// unit & equipment number ---------------------------------------------------
      L     DB1400.DBW    0;
      T     #UnitNo;

      L     DB1405.DBW   14;
      L     1000;
      *I    ;
      L     #UnitNo;
      +I    ;
      T     #EquipmentID;

// CIP ----------------------------------------------------------------------
      L     DB1405.DBW   18;
      L     0;
      <I    ;
      =     #CIP;

// Communicating Units-------------------------------------------------------
      L     DB1405.DBD   10;
      L     DB1405.DBD  106;
      ==D   ;
      =     #ComCIP;

// emergency OK -------------------------------------------------------------
      A     DB1405.DBX   75.0; //General Emergency Stop OK
      =     #EStopOK;

NETWORK
TITLE =read other unit's data

      SET   ;

// ... General Unit ----------/

      CALL FC   563 (
           ActReq                   := M    101.0,
           PLCNo                    := DB1405.DBW   14,
           SourceUnitNo             := 99,
           IsTUnit                  := FALSE,
           DstComDRec               := DB1405.GEN,

           RET_VAL                  := #wRetVal);

// ... CIP Unit ------------- /

      CALL FC   563 (
           ActReq                   := M    101.0,
           PLCNo                    := 1,
           SourceUnitNo             := 71,
           IsTUnit                  := FALSE,
           DstComDRec               := DB1405.CIP,

           RET_VAL                  := #wRetVal);


NETWORK
TITLE =remote start

      SET   ;
// !!! insert correct condition of unit start !!!
      A     DB1401.DBX   15.0;
      A     DB1401.DBX   17.4;
      CLR   ;
      JCN   Strt;
      L     DB1405.DBD   10;
//L        L#-1;                            // Prid negative to start on its own
      T     #Prid;

      CALL FC    48 (
           UnitNo                   := #UnitNo,
           PrId                     := #Prid,
           Run                      := DB1401.DBX   17.4,
           PrIdTransfer             := TRUE,
           Start                    := TRUE,
           RetVal                   := #wRetVal);
Strt: NOP   0;
NETWORK
TITLE =external releases

      SET   ;
NETWORK
TITLE =write own unit data

      SET   ;

//-- CIP Communication ---------------------------------------
      AN    DB1401.DBX   15.0;
//      AN "U040SeqD".Seq.PO.B30 // CIP Active (Slave)
      A     #ComCIP;
      JCN   NCIP;
//Conductivity CIP Return
      L     DB1405.DBD  150;
      T     DB1401.DBD  626;

//Temperature CIP Return
      L     DB1405.DBD  146;
      T     DB1401.DBD  594;

//CIP Prerun Pump SP

      CALL FC    45 (
           SFM                      := DB1401.DBD  686,

           Indexes                  := #SFM36);

      L     0.000000e+000;
      A     #SFM36.I01;
      =     DB1405.DBX  171.7;
      JCN   pfc;
      L     DB1401.DBD  654;
pfc:  NOP   0;
      A     #SFM36.I02;
      =     DB1405.DBX  172.0;
      JCN   ppc;
      L     DB1401.DBD  670;
ppc:  NOP   0;
      A     #SFM36.I03;
      =     DB1405.DBX  171.6;
      JCN   pxc;
      L     DB1401.DBD  574;
pxc:  NOP   0;
      T     DB1405.DBD  182;

//CIP Return
      L     DB1401.DBD  558;
      T     DB1405.DBD  186;
      L     DB1405.DBD  138;
      T     DB1401.DBD  562;

//CIP Prerun
      L     DB1401.DBD  542;
      T     DB1405.DBD  190;
      L     DB1405.DBD  142;
      T     DB1401.DBD  546;

// Write Own Data to CIP
      L     DB1405.DBD   10;
      T     DB1405.DBD  154;

      L     DB1405.DBW   14;
      T     DB1405.DBW  158;

      L     DB1405.DBW   16;
      T     DB1405.DBW  160;

      L     DB1405.DBW   18;
      T     DB1405.DBW  162;

      L     DB1405.DBW   20;
      T     DB1405.DBW  164;

      L     DB1405.DBW   22;
      T     DB1405.DBW  166;

      A     DB1405.DBX   24.0;
      =     DB1405.DBX  168.0;

      A     DB1405.DBX   24.1;
      =     DB1405.DBX  168.1;

      A     DB1405.DBX   24.2;
      =     DB1405.DBX  168.2;

      A     DB1405.DBX   24.3;
      =     DB1405.DBX  168.3;

      A     DB1405.DBX   24.4;
      =     DB1405.DBX  168.4;

      A     DB1405.DBX   24.5;
      =     DB1405.DBX  168.5;

      A     DB1405.DBX   24.6;
      =     DB1405.DBX  168.6;

      A     DB1405.DBX   24.7;
      =     DB1405.DBX  168.7;

// Copy Data to CIP
      CALL SFC   20 (
           SRCBLK                   := DB1405.ToCIP,
           RET_VAL                  := #iRetVal,
           DSTBLK                   := DB1405.ToCIP);

NCIP: NOP   0;

//Empty Signal
//A     "U040SpID".SpI.Sig //!!!! Insert correct Empty Signal !!!
      CLR   ;
      =     DB1405.DBX   26.5;

//Full Signal
//A     "U040SpID".SpI.Sig //!!!! Insert correct Full Signal !!!
      CLR   ;
      =     DB1405.DBX   26.2;

//CIP Program Selected
      A     #CIP;
      =     DB1405.DBX   27.1;

// Emergency Stop
      A     #EStopOK; //If needed add or replace with own SpI
      =     DB1405.DBX   27.0; //Emergency Stop OK


NETWORK
TITLE = read from other unit data

END_FUNCTION_BLOCK

FUNCTION_BLOCK FB 1409
TITLE =U040: Water Treatment General
AUTHOR : Woermann
FAMILY : BOTEC_F1
NAME : Sim
VERSION : 0.1


VAR_TEMP
  CIP : BOOL ;	//CIP active
  xTmp : BOOL ;	//Temporary BOOL (free for general use)
  iTmp : INT ;	//Temporary INT (free for general use)
  rTmp : REAL ;	//Temporary REAL (free for general use)
  UnitNo : INT ;	//Unit Number
END_VAR
BEGIN
NETWORK
TITLE =General

      SET   ;
// get unit number ----------------------------------------------------------
      L     DB1400.DBW    0;
      T     #UnitNo;

// CIP ----------------------------------------------------------------------
      L     DB1401.DBD   54;
      L     0;
      <D    ;
      =     #CIP;

NETWORK
TITLE =Actuator

      A     DB1401.DBX   17.3;

NETWORK
TITLE =Special Input

      A     DB1401.DBX   17.3;
      =     DB2401.DBX   81.3;
      =     DB2401.DBX  141.3;
      =     DB2401.DBX  201.3;
      =     DB2401.DBX  261.3;
      =     DB2401.DBX  321.3;
      =     DB2401.DBX  381.3;

NETWORK
TITLE =Counter

      A     DB1401.DBX   17.3;
      A     M    101.0;


      CLR   ;
NETWORK
TITLE =Analog Input

      A     DB1401.DBX   17.3;

NETWORK
TITLE =Universal Value

      A     DB1401.DBX   17.3;
//      =     "U040UnVD".unv001.Sim;
//      =     "U040UnVD".unv002.Sim;

NETWORK
TITLE =PID

      A     DB1401.DBX   17.3;

NETWORK
TITLE =Message

      A     DB1401.DBX   17.3;
//      =     "U040MsgD".msg001.Sim;
//      =     "U040MsgD".msg002.Sim;

NETWORK
TITLE =VLT

      A     DB1401.DBX   17.3;

END_FUNCTION_BLOCK

FUNCTION_BLOCK FB 1435
TITLE =U043: Water Transfer Plant 3
FAMILY : BOTEC_F1
NAME : Comm
VERSION : 0.1


VAR_TEMP
  iRetVal : INT ;	//return value as integer
  wRetVal : WORD ;	//return value as word
  Run : BOOL ;	//Unit in "RUN" mode
  EStopOK : BOOL ;	//Emergency Stop OK
  CIP : BOOL ;	//CIP Program Selected
  ComCIP : BOOL ;	//Communication with CIP Active
  xTmp : BOOL ;	//Temporary BOOL (free for general use)
  iTmp : INT ;	//Temporary INT (free for general use)
  rTmp : REAL ;	//Temporary REAL (free for general use)
  dTmp : DINT ;	//Temporary DINT (free for general use)
  UnitNo : INT ;	//Unit Number
  EquipmentID : INT ;	//Equipment ID
  Prid : DINT ;	//Process ID
  SFM36 : STRUCT 	// CIP Pump Mode
   I00 : BOOL ;	// Off
   I01 : BOOL ;	// Flow
   I02 : BOOL ;	// Pressure
   I03 : BOOL ;	// Fix Speed
   I04 : BOOL ;
   I05 : BOOL ;
   I06 : BOOL ;
   I07 : BOOL ;
   I08 : BOOL ;
   I09 : BOOL ;
   I10 : BOOL ;
   I11 : BOOL ;
   I12 : BOOL ;
   I13 : BOOL ;
   I14 : BOOL ;
   I15 : BOOL ;
   I16 : BOOL ;
   I17 : BOOL ;
   I18 : BOOL ;
   I19 : BOOL ;
   I20 : BOOL ;
   I21 : BOOL ;
   I22 : BOOL ;
   I23 : BOOL ;
   I24 : BOOL ;
   I25 : BOOL ;
   I26 : BOOL ;
   I27 : BOOL ;
   I28 : BOOL ;
   I29 : BOOL ;
   I30 : BOOL ;
   I31 : BOOL ;
  END_STRUCT ;
END_VAR
BEGIN
NETWORK
TITLE =general

      SET   ;

// unit & equipment number ---------------------------------------------------
      L     DB1430.DBW    0;
      T     #UnitNo;

      L     DB1435.DBW   14;
      L     1000;
      *I    ;
      L     #UnitNo;
      +I    ;
      T     #EquipmentID;

// CIP ----------------------------------------------------------------------
      L     DB1435.DBW   18;
      L     0;
      <I    ;
      =     #CIP;

// Communicating Units-------------------------------------------------------
      L     DB1435.DBD   10;
      L     DB1435.DBD  106;
      ==D   ;
      =     #ComCIP;

// emergency OK -------------------------------------------------------------
      A     DB1435.DBX   75.0; //General Emergency Stop OK
      =     #EStopOK;

NETWORK
TITLE =read other unit's data

      SET   ;

// ... General Unit ----------/

      CALL FC   563 (
           ActReq                   := M    101.0,
           PLCNo                    := DB1435.DBW   14,
           SourceUnitNo             := 99,
           IsTUnit                  := FALSE,
           DstComDRec               := DB1435.GEN,
           RET_VAL                  := #wRetVal);


// ... CIP Unit ------------- /

      CALL FC   563 (
           ActReq                   := M    101.0,
           PLCNo                    := 1,
           SourceUnitNo             := 71,
           IsTUnit                  := FALSE,
           DstComDRec               := DB1435.CIP,
           RET_VAL                  := #wRetVal);



NETWORK
TITLE =remote start

      SET   ;
// !!! insert correct condition of unit start !!!
      A     DB1431.DBX   15.0;
      A     DB1431.DBX   17.4;
      CLR   ;
      JCN   Strt;
      L     L#-1; // Prid negative to start on its own
      T     #Prid;

      CALL FC    48 (
           UnitNo                   := #UnitNo,
           PrId                     := #Prid,
           Run                      := DB1431.DBX   17.4,
           PrIdTransfer             := TRUE,
           Start                    := TRUE,
           RetVal                   := #wRetVal);
Strt: NOP   0;
NETWORK
TITLE =external releases

      SET   ;
      =     DB2430.DBX  186.7;
      =     DB2430.DBX  266.7;
      =     DB2430.DBX  346.7;
NETWORK
TITLE =write own unit data

      SET   ;

//-- CIP Communication ---------------------------------------
      AN    DB1431.DBX   15.0;
//      AN "U043SeqD".Seq.PO.B30 // CIP Active (Slave)
      A     #ComCIP;
      JCN   NCIP;
//Conductivity CIP Return
      L     DB1435.DBD  150;
      T     DB1431.DBD  626;

//Temperature CIP Return
      L     DB1435.DBD  146;
      T     DB1431.DBD  594;

//CIP Prerun Pump SP

      CALL FC    45 (
           SFM                      := DB1431.DBD  686,
           Indexes                  := #SFM36);


      L     0.000000e+000;
      A     #SFM36.I01;
      =     DB1435.DBX  171.7;
      JCN   pfc;
      L     DB1431.DBD  654;
pfc:  NOP   0;
      A     #SFM36.I02;
      =     DB1435.DBX  172.0;
      JCN   ppc;
      L     DB1431.DBD  670;
ppc:  NOP   0;
      A     #SFM36.I03;
      =     DB1435.DBX  171.6;
      JCN   pxc;
      L     DB1431.DBD  574;
pxc:  NOP   0;
      T     DB1435.DBD  182;

//CIP Return
      L     DB1431.DBD  558;
      T     DB1435.DBD  186;
      L     DB1435.DBD  138;
      T     DB1431.DBD  562;

//CIP Prerun
      L     DB1431.DBD  542;
      T     DB1435.DBD  190;
      L     DB1435.DBD  142;
      T     DB1431.DBD  546;

// Write Own Data to CIP
      L     DB1435.DBD   10;
      T     DB1435.DBD  154;

      L     DB1435.DBW   14;
      T     DB1435.DBW  158;

      L     DB1435.DBW   16;
      T     DB1435.DBW  160;

      L     DB1435.DBW   18;
      T     DB1435.DBW  162;

      L     DB1435.DBW   20;
      T     DB1435.DBW  164;

      L     DB1435.DBW   22;
      T     DB1435.DBW  166;

      A     DB1435.DBX   24.0;
      =     DB1435.DBX  168.0;

      A     DB1435.DBX   24.1;
      =     DB1435.DBX  168.1;

      A     DB1435.DBX   24.2;
      =     DB1435.DBX  168.2;

      A     DB1435.DBX   24.3;
      =     DB1435.DBX  168.3;

      A     DB1435.DBX   24.4;
      =     DB1435.DBX  168.4;

      A     DB1435.DBX   24.5;
      =     DB1435.DBX  168.5;

      A     DB1435.DBX   24.6;
      =     DB1435.DBX  168.6;

      A     DB1435.DBX   24.7;
      =     DB1435.DBX  168.7;

// Copy Data to CIP
      CALL SFC   20 (
           SRCBLK                   := DB1435.ToCIP,
           RET_VAL                  := #iRetVal,
           DSTBLK                   := DB1435.ToCIP);

NCIP: NOP   0;

//Empty Signal
//A     "U043SpID".SpI.Sig //!!!! Insert correct Empty Signal !!!
      CLR   ;
      =     DB1435.DBX   26.5;

//Full Signal
//A     "U043SpID".SpI.Sig //!!!! Insert correct Full Signal !!!
      CLR   ;
      =     DB1435.DBX   26.2;

//CIP Program Selected
      A     #CIP;
      =     DB1435.DBX   27.1;

// Emergency Stop
      A     #EStopOK; //If needed add or replace with own SpI
      =     DB1435.DBX   27.0; //Emergency Stop OK



NETWORK
TITLE = read from other unit data



END_FUNCTION_BLOCK

FUNCTION_BLOCK FB 1439
TITLE =U043: Water Transfer Plant 3
AUTHOR : Woermann
FAMILY : BOTEC_F1
NAME : Sim
VERSION : 0.1


VAR_TEMP
  CIP : BOOL ;	//CIP active
  xTmp : BOOL ;	//Temporary BOOL (free for general use)
  iTmp : INT ;	//Temporary INT (free for general use)
  rTmp : REAL ;	//Temporary REAL (free for general use)
  UnitNo : INT ;	//Unit Number
END_VAR
BEGIN
NETWORK
TITLE =General

      SET   ;
// get unit number ----------------------------------------------------------
      L     DB1430.DBW    0;
      T     #UnitNo;

// CIP ----------------------------------------------------------------------
      L     DB1431.DBD   54;
      L     0;
      <D    ;
      =     #CIP;

NETWORK
TITLE =Actuator

      A     DB1431.DBX   17.3;
      =     DB2430.DBX  185.3;
      =     DB2430.DBX  265.3;
      =     DB2430.DBX  345.3;

NETWORK
TITLE =Special Input

      A     DB1431.DBX   17.3;
      =     DB2431.DBX   81.3;

NETWORK
TITLE =Counter

      A     DB1431.DBX   17.3;
      A     M    101.0;


      CLR   ;
NETWORK
TITLE =Analog Input

      A     DB1431.DBX   17.3;

NETWORK
TITLE =Universal Value

      A     DB1431.DBX   17.3;
//      =     "U043UnVD".unv001.Sim;
//      =     "U043UnVD".unv002.Sim;
//      =     "U043UnVD".unv003.Sim;
//      =     "U043UnVD".unv004.Sim;

NETWORK
TITLE =PID

      A     DB1431.DBX   17.3;

NETWORK
TITLE =Message

      A     DB1431.DBX   17.3;
//      =     "U043MsgD".msg001.Sim;
//      =     "U043MsgD".msg002.Sim;
//      =     "U043MsgD".msg003.Sim;

NETWORK
TITLE =VLT

      A     DB1431.DBX   17.3;

END_FUNCTION_BLOCK

FUNCTION_BLOCK FB 1455
TITLE =U045: Water Transfer Plant 5
FAMILY : BOTEC_F1
NAME : Comm
VERSION : 0.1


VAR_TEMP
  iRetVal : INT ;	//return value as integer
  wRetVal : WORD ;	//return value as word
  Run : BOOL ;	//Unit in "RUN" mode
  EStopOK : BOOL ;	//Emergency Stop OK
  CIP : BOOL ;	//CIP Program Selected
  ComCIP : BOOL ;	//Communication with CIP Active
  xTmp : BOOL ;	//Temporary BOOL (free for general use)
  iTmp : INT ;	//Temporary INT (free for general use)
  rTmp : REAL ;	//Temporary REAL (free for general use)
  dTmp : DINT ;	//Temporary DINT (free for general use)
  UnitNo : INT ;	//Unit Number
  EquipmentID : INT ;	//Equipment ID
  Prid : DINT ;	//Process ID
  SFM36 : STRUCT 	// CIP Pump Mode
   I00 : BOOL ;	// Off
   I01 : BOOL ;	// Flow
   I02 : BOOL ;	// Pressure
   I03 : BOOL ;	// Fix Speed
   I04 : BOOL ;
   I05 : BOOL ;
   I06 : BOOL ;
   I07 : BOOL ;
   I08 : BOOL ;
   I09 : BOOL ;
   I10 : BOOL ;
   I11 : BOOL ;
   I12 : BOOL ;
   I13 : BOOL ;
   I14 : BOOL ;
   I15 : BOOL ;
   I16 : BOOL ;
   I17 : BOOL ;
   I18 : BOOL ;
   I19 : BOOL ;
   I20 : BOOL ;
   I21 : BOOL ;
   I22 : BOOL ;
   I23 : BOOL ;
   I24 : BOOL ;
   I25 : BOOL ;
   I26 : BOOL ;
   I27 : BOOL ;
   I28 : BOOL ;
   I29 : BOOL ;
   I30 : BOOL ;
   I31 : BOOL ;
  END_STRUCT ;
  SRCUnit : INT ;	//Source Water Tank
  DummyBool : BOOL ;
END_VAR
BEGIN
NETWORK
TITLE =general

      SET   ;

// unit & equipment number ---------------------------------------------------
      L     DB1450.DBW    0;
      T     #UnitNo;

      L     DB1455.DBW   14;
      L     1000;
      *I    ;
      L     #UnitNo;
      +I    ;
      T     #EquipmentID;

// CIP ----------------------------------------------------------------------
      L     DB1455.DBW   18;
      L     0;
      <I    ;
      =     #CIP;

// Communicating Units-------------------------------------------------------
      L     DB1455.DBD   10;
      L     DB1455.DBD  106;
      ==D   ;
      =     #ComCIP;

// emergency OK -------------------------------------------------------------
      A     DB1455.DBX   75.0; //General Emergency Stop OK
      =     #EStopOK;

NETWORK
TITLE =remote start

      SET   ;
      L     DB1455.DBD   10;

// !!! insert correct condition of unit start !!!
      A     DB1451.DBX   15.0;
      A     DB1451.DBX   17.4;
      CLR   ;
      JCN   Strt;
      L     DB1455.DBD   10;
//L        L#-1;                            // Prid negative to start on its own
      T     #Prid;

      CALL FC    48 (
           UnitNo                   := #UnitNo,
           PrId                     := #Prid,
           Run                      := DB1451.DBX   17.4,
           PrIdTransfer             := TRUE,
           Start                    := TRUE,
           RetVal                   := #wRetVal);
Strt: NOP   0;
END_FUNCTION_BLOCK

FUNCTION_BLOCK FB 1459
TITLE =U045: Water Transfer Plant 5
AUTHOR : Woermann
FAMILY : BOTEC_F1
NAME : Sim
VERSION : 0.1


VAR_TEMP
  CIP : BOOL ;	//CIP active
  xTmp : BOOL ;	//Temporary BOOL (free for general use)
  iTmp : INT ;	//Temporary INT (free for general use)
  rTmp : REAL ;	//Temporary REAL (free for general use)
  UnitNo : INT ;	//Unit Number
END_VAR
BEGIN
NETWORK
TITLE =General

      SET   ;
// get unit number ----------------------------------------------------------
      L     DB1450.DBW    0;
      T     #UnitNo;

// CIP ----------------------------------------------------------------------
      L     DB1451.DBD   54;
      L     0;
      <D    ;
      =     #CIP;

NETWORK
TITLE =Actuator

      A     DB1451.DBX   17.3;
      =     DB2450.DBX  425.3;
      =     DB2450.DBX  505.3;
      =     DB2450.DBX  585.3;
      =     DB2450.DBX  665.3;

NETWORK
TITLE =Special Input

      A     DB1451.DBX   17.3;

NETWORK
TITLE =Counter

      A     DB1451.DBX   17.3;
      A     M    101.0;


      CLR   ;
NETWORK
TITLE =Analog Input

      A     DB1451.DBX   17.3;

NETWORK
TITLE =Universal Value

      A     DB1451.DBX   17.3;
//      =     "U045UnVD".unv001.Sim;
//      =     "U045UnVD".unv002.Sim;
//      =     "U045UnVD".unv003.Sim;
//      =     "U045UnVD".unv004.Sim;

NETWORK
TITLE =PID

      A     DB1451.DBX   17.3;

NETWORK
TITLE =Message

      A     DB1451.DBX   17.3;
//      =     "U045MsgD".msg001.Sim;
//      =     "U045MsgD".msg002.Sim;
//      =     "U045MsgD".msg003.Sim;

NETWORK
TITLE =VLT

      A     DB1451.DBX   17.3;

END_FUNCTION_BLOCK

FUNCTION_BLOCK FB 1475
TITLE =U047: Water Transfer Plant 7
FAMILY : BOTEC_F1
NAME : Comm
VERSION : 0.1


VAR_TEMP
  iRetVal : INT ;	//return value as integer
  wRetVal : WORD ;	//return value as word
  Run : BOOL ;	//Unit in "RUN" mode
  EStopOK : BOOL ;	//Emergency Stop OK
  CIP : BOOL ;	//CIP Program Selected
  ComCIP : BOOL ;	//Communication with CIP Active
  xTmp : BOOL ;	//Temporary BOOL (free for general use)
  iTmp : INT ;	//Temporary INT (free for general use)
  rTmp : REAL ;	//Temporary REAL (free for general use)
  dTmp : DINT ;	//Temporary DINT (free for general use)
  UnitNo : INT ;	//Unit Number
  EquipmentID : INT ;	//Equipment ID
  Prid : DINT ;	//Process ID
  SFM36 : STRUCT 	// CIP Pump Mode
   I00 : BOOL ;	// Off
   I01 : BOOL ;	// Flow
   I02 : BOOL ;	// Pressure
   I03 : BOOL ;	// Fix Speed
   I04 : BOOL ;
   I05 : BOOL ;
   I06 : BOOL ;
   I07 : BOOL ;
   I08 : BOOL ;
   I09 : BOOL ;
   I10 : BOOL ;
   I11 : BOOL ;
   I12 : BOOL ;
   I13 : BOOL ;
   I14 : BOOL ;
   I15 : BOOL ;
   I16 : BOOL ;
   I17 : BOOL ;
   I18 : BOOL ;
   I19 : BOOL ;
   I20 : BOOL ;
   I21 : BOOL ;
   I22 : BOOL ;
   I23 : BOOL ;
   I24 : BOOL ;
   I25 : BOOL ;
   I26 : BOOL ;
   I27 : BOOL ;
   I28 : BOOL ;
   I29 : BOOL ;
   I30 : BOOL ;
   I31 : BOOL ;
  END_STRUCT ;
END_VAR
BEGIN
NETWORK
TITLE =general

      SET   ;

// unit & equipment number ---------------------------------------------------
      L     DB1470.DBW    0;
      T     #UnitNo;

      L     DB1475.DBW   14;
      L     1000;
      *I    ;
      L     #UnitNo;
      +I    ;
      T     #EquipmentID;

// CIP ----------------------------------------------------------------------
      L     DB1475.DBW   18;
      L     0;
      <I    ;
      =     #CIP;

// Communicating Units-------------------------------------------------------
      L     DB1475.DBD   10;
      L     DB1475.DBD  106;
      ==D   ;
      =     #ComCIP;

// emergency OK -------------------------------------------------------------
      A     DB1475.DBX   75.0; //General Emergency Stop OK
      =     #EStopOK;

NETWORK
TITLE =read other unit's data

      SET   ;

// ... General Unit ----------/

      CALL FC   563 (
           ActReq                   := M    101.0,
           PLCNo                    := DB1475.DBW   14,
           SourceUnitNo             := 99,
           IsTUnit                  := FALSE,
           DstComDRec               := DB1475.GEN,
           RET_VAL                  := #wRetVal);


NETWORK
TITLE =remote start

      SET   ;
// !!! insert correct condition of unit start !!!
      A     DB1471.DBX   15.0;
      A     DB1471.DBX   17.4;
      CLR   ;
      JCN   Strt;
      L     DB1475.DBD   10;
//L        L#-1;                            // Prid negative to start on its own
      T     #Prid;

      CALL FC    48 (
           UnitNo                   := #UnitNo,
           PrId                     := #Prid,
           Run                      := DB1471.DBX   17.4,
           PrIdTransfer             := TRUE,
           Start                    := TRUE,
           RetVal                   := #wRetVal);
Strt: NOP   0;
NETWORK
TITLE =external releases

      SET   ;
      =     DB2470.DBX  186.7;
      =     DB2470.DBX  266.7;
      =     DB2470.DBX  346.7;
      =     DB2470.DBX  426.7;
      =     DB2470.DBX  506.7;
      =     DB2470.DBX  586.7;
      =     DB2470.DBX  666.7;
NETWORK
TITLE =write own unit data

      SET   ;

//-- CIP Communication ---------------------------------------
      AN    DB1471.DBX   15.0;
//      AN "U047SeqD".Seq.PO.B30 // CIP Active (Slave)
      A     #ComCIP;
      JCN   NCIP;
//Conductivity CIP Return
      L     DB1475.DBD  150;
      T     DB1471.DBD  626;

//Temperature CIP Return
      L     DB1475.DBD  146;
      T     DB1471.DBD  594;

//CIP Prerun Pump SP

      CALL FC    45 (
           SFM                      := DB1471.DBD  686,
           Indexes                  := #SFM36);


      L     0.000000e+000;
      A     #SFM36.I01;
      =     DB1475.DBX  171.7;
      JCN   pfc;
      L     DB1471.DBD  654;
pfc:  NOP   0;
      A     #SFM36.I02;
      =     DB1475.DBX  172.0;
      JCN   ppc;
      L     DB1471.DBD  670;
ppc:  NOP   0;
      A     #SFM36.I03;
      =     DB1475.DBX  171.6;
      JCN   pxc;
      L     DB1471.DBD  574;
pxc:  NOP   0;
      T     DB1475.DBD  182;

//CIP Return
      L     DB1471.DBD  558;
      T     DB1475.DBD  186;
      L     DB1475.DBD  138;
      T     DB1471.DBD  562;

//CIP Prerun
      L     DB1471.DBD  542;
      T     DB1475.DBD  190;
      L     DB1475.DBD  142;
      T     DB1471.DBD  546;

// Write Own Data to CIP
      L     DB1475.DBD   10;
      T     DB1475.DBD  154;

      L     DB1475.DBW   14;
      T     DB1475.DBW  158;

      L     DB1475.DBW   16;
      T     DB1475.DBW  160;

      L     DB1475.DBW   18;
      T     DB1475.DBW  162;

      L     DB1475.DBW   20;
      T     DB1475.DBW  164;

      L     DB1475.DBW   22;
      T     DB1475.DBW  166;

      A     DB1475.DBX   24.0;
      =     DB1475.DBX  168.0;

      A     DB1475.DBX   24.1;
      =     DB1475.DBX  168.1;

      A     DB1475.DBX   24.2;
      =     DB1475.DBX  168.2;

      A     DB1475.DBX   24.3;
      =     DB1475.DBX  168.3;

      A     DB1475.DBX   24.4;
      =     DB1475.DBX  168.4;

      A     DB1475.DBX   24.5;
      =     DB1475.DBX  168.5;

      A     DB1475.DBX   24.6;
      =     DB1475.DBX  168.6;

      A     DB1475.DBX   24.7;
      =     DB1475.DBX  168.7;

// Copy Data to CIP
      CALL SFC   20 (
           SRCBLK                   := DB1475.ToCIP,
           RET_VAL                  := #iRetVal,
           DSTBLK                   := DB1475.ToCIP);

NCIP: NOP   0;

//Empty Signal
//A     "U047SpID".SpI.Sig //!!!! Insert correct Empty Signal !!!
      CLR   ;
      =     DB1475.DBX   26.5;

//Full Signal
//A     "U047SpID".SpI.Sig //!!!! Insert correct Full Signal !!!
      CLR   ;
      =     DB1475.DBX   26.2;

//CIP Program Selected
      A     #CIP;
      =     DB1475.DBX   27.1;

// Emergency Stop
      A     #EStopOK; //If needed add or replace with own SpI
      =     DB1475.DBX   27.0; //Emergency Stop OK


NETWORK
TITLE = read from other unit data



END_FUNCTION_BLOCK

FUNCTION_BLOCK FB 1479
TITLE =U047: Water Transfer Plant 7
AUTHOR : Woermann
FAMILY : BOTEC_F1
NAME : Sim
VERSION : 0.1


VAR_TEMP
  CIP : BOOL ;	//CIP active
  xTmp : BOOL ;	//Temporary BOOL (free for general use)
  iTmp : INT ;	//Temporary INT (free for general use)
  rTmp : REAL ;	//Temporary REAL (free for general use)
  UnitNo : INT ;	//Unit Number
END_VAR
BEGIN
NETWORK
TITLE =General

      SET   ;
// get unit number ----------------------------------------------------------
      L     DB1470.DBW    0;
      T     #UnitNo;

// CIP ----------------------------------------------------------------------
      L     DB1471.DBD   54;
      L     0;
      <D    ;
      =     #CIP;

NETWORK
TITLE =Actuator

      A     DB1471.DBX   17.3;
      =     DB2470.DBX  185.3;
      =     DB2470.DBX  265.3;
      =     DB2470.DBX  345.3;
      =     DB2470.DBX  425.3;
      =     DB2470.DBX  505.3;
      =     DB2470.DBX  585.3;
      =     DB2470.DBX  665.3;

NETWORK
TITLE =Special Input

      A     DB1471.DBX   17.3;

NETWORK
TITLE =Counter

      A     DB1471.DBX   17.3;
      A     M    101.0;


      CLR   ;
NETWORK
TITLE =Analog Input

      A     DB1471.DBX   17.3;

NETWORK
TITLE =Universal Value

      A     DB1471.DBX   17.3;
//      =     "U047UnVD".unv001.Sim;
//      =     "U047UnVD".unv002.Sim;
//      =     "U047UnVD".unv003.Sim;
//      =     "U047UnVD".unv004.Sim;

NETWORK
TITLE =PID

      A     DB1471.DBX   17.3;

NETWORK
TITLE =Message

      A     DB1471.DBX   17.3;
//      =     "U047MsgD".msg001.Sim;
//      =     "U047MsgD".msg002.Sim;
//      =     "U047MsgD".msg003.Sim;

NETWORK
TITLE =VLT

      A     DB1471.DBX   17.3;

END_FUNCTION_BLOCK

FUNCTION_BLOCK FB 1485
TITLE =U048: Water Transfer Plant 8
FAMILY : BOTEC_F1
NAME : Comm
VERSION : 0.1


VAR_TEMP
  iRetVal : INT ;	//return value as integer
  wRetVal : WORD ;	//return value as word
  Run : BOOL ;	//Unit in "RUN" mode
  EStopOK : BOOL ;	//Emergency Stop OK
  CIP : BOOL ;	//CIP Program Selected
  ComCIP : BOOL ;	//Communication with CIP Active
  xTmp : BOOL ;	//Temporary BOOL (free for general use)
  iTmp : INT ;	//Temporary INT (free for general use)
  rTmp : REAL ;	//Temporary REAL (free for general use)
  dTmp : DINT ;	//Temporary DINT (free for general use)
  UnitNo : INT ;	//Unit Number
  EquipmentID : INT ;	//Equipment ID
  Prid : DINT ;	//Process ID
  SFM36 : STRUCT 	// CIP Pump Mode
   I00 : BOOL ;	// Off
   I01 : BOOL ;	// Flow
   I02 : BOOL ;	// Pressure
   I03 : BOOL ;	// Fix Speed
   I04 : BOOL ;
   I05 : BOOL ;
   I06 : BOOL ;
   I07 : BOOL ;
   I08 : BOOL ;
   I09 : BOOL ;
   I10 : BOOL ;
   I11 : BOOL ;
   I12 : BOOL ;
   I13 : BOOL ;
   I14 : BOOL ;
   I15 : BOOL ;
   I16 : BOOL ;
   I17 : BOOL ;
   I18 : BOOL ;
   I19 : BOOL ;
   I20 : BOOL ;
   I21 : BOOL ;
   I22 : BOOL ;
   I23 : BOOL ;
   I24 : BOOL ;
   I25 : BOOL ;
   I26 : BOOL ;
   I27 : BOOL ;
   I28 : BOOL ;
   I29 : BOOL ;
   I30 : BOOL ;
   I31 : BOOL ;
  END_STRUCT ;
END_VAR
BEGIN
NETWORK
TITLE =general

      SET   ;

// unit & equipment number ---------------------------------------------------
      L     DB1480.DBW    0;
      T     #UnitNo;

      L     DB1485.DBW   14;
      L     1000;
      *I    ;
      L     #UnitNo;
      +I    ;
      T     #EquipmentID;

// CIP ----------------------------------------------------------------------
      L     DB1485.DBW   18;
      L     0;
      <I    ;
      =     #CIP;

// Communicating Units-------------------------------------------------------
      L     DB1485.DBD   10;
      L     DB1485.DBD  106;
      ==D   ;
      =     #ComCIP;

// emergency OK -------------------------------------------------------------
      A     DB1485.DBX   75.0; //General Emergency Stop OK
      =     #EStopOK;

NETWORK
TITLE =read other unit's data

      SET   ;

// ... General Unit ----------/

      CALL FC   563 (
           ActReq                   := M    101.0,
           PLCNo                    := DB1485.DBW   14,
           SourceUnitNo             := 99,
           IsTUnit                  := FALSE,
           DstComDRec               := DB1485.GEN,
           RET_VAL                  := #wRetVal);

NETWORK
TITLE =remote start

      SET   ;
// !!! insert correct condition of unit start !!!
      A     DB1481.DBX   15.0;
      A     DB1481.DBX   17.4;
      CLR   ;
      JCN   Strt;
      L     DB1485.DBD   10;
//L        L#-1;                            // Prid negative to start on its own
      T     #Prid;

      CALL FC    48 (
           UnitNo                   := #UnitNo,
           PrId                     := #Prid,
           Run                      := DB1481.DBX   17.4,
           PrIdTransfer             := TRUE,
           Start                    := TRUE,
           RetVal                   := #wRetVal);
Strt: NOP   0;
NETWORK
TITLE =external releases

      SET   ;
      =     DB2480.DBX  426.7;
      =     DB2480.DBX  506.7;
      =     DB2480.DBX  586.7;
      =     DB2480.DBX  666.7;
NETWORK
TITLE =write own unit data

      SET   ;

//-- CIP Communication ---------------------------------------
      AN    DB1481.DBX   15.0;
//      AN "U048SeqD".Seq.PO.B30 // CIP Active (Slave)
      A     #ComCIP;
      JCN   NCIP;
//Conductivity CIP Return
      L     DB1485.DBD  150;
      T     DB1481.DBD  626;

//Temperature CIP Return
      L     DB1485.DBD  146;
      T     DB1481.DBD  594;

//CIP Prerun Pump SP

      CALL FC    45 (
           SFM                      := DB1481.DBD  686,
           Indexes                  := #SFM36);


      L     0.000000e+000;
      A     #SFM36.I01;
      =     DB1485.DBX  171.7;
      JCN   pfc;
      L     DB1481.DBD  654;
pfc:  NOP   0;
      A     #SFM36.I02;
      =     DB1485.DBX  172.0;
      JCN   ppc;
      L     DB1481.DBD  670;
ppc:  NOP   0;
      A     #SFM36.I03;
      =     DB1485.DBX  171.6;
      JCN   pxc;
      L     DB1481.DBD  574;
pxc:  NOP   0;
      T     DB1485.DBD  182;

//CIP Return
      L     DB1481.DBD  558;
      T     DB1485.DBD  186;
      L     DB1485.DBD  138;
      T     DB1481.DBD  562;

//CIP Prerun
      L     DB1481.DBD  542;
      T     DB1485.DBD  190;
      L     DB1485.DBD  142;
      T     DB1481.DBD  546;

// Write Own Data to CIP
      L     DB1485.DBD   10;
      T     DB1485.DBD  154;

      L     DB1485.DBW   14;
      T     DB1485.DBW  158;

      L     DB1485.DBW   16;
      T     DB1485.DBW  160;

      L     DB1485.DBW   18;
      T     DB1485.DBW  162;

      L     DB1485.DBW   20;
      T     DB1485.DBW  164;

      L     DB1485.DBW   22;
      T     DB1485.DBW  166;

      A     DB1485.DBX   24.0;
      =     DB1485.DBX  168.0;

      A     DB1485.DBX   24.1;
      =     DB1485.DBX  168.1;

      A     DB1485.DBX   24.2;
      =     DB1485.DBX  168.2;

      A     DB1485.DBX   24.3;
      =     DB1485.DBX  168.3;

      A     DB1485.DBX   24.4;
      =     DB1485.DBX  168.4;

      A     DB1485.DBX   24.5;
      =     DB1485.DBX  168.5;

      A     DB1485.DBX   24.6;
      =     DB1485.DBX  168.6;

      A     DB1485.DBX   24.7;
      =     DB1485.DBX  168.7;

// Copy Data to CIP
      CALL SFC   20 (
           SRCBLK                   := DB1485.ToCIP,
           RET_VAL                  := #iRetVal,
           DSTBLK                   := DB1485.ToCIP);

NCIP: NOP   0;

//Empty Signal
//A     "U048SpID".SpI.Sig //!!!! Insert correct Empty Signal !!!
      CLR   ;
      =     DB1485.DBX   26.5;

//Full Signal
//A     "U048SpID".SpI.Sig //!!!! Insert correct Full Signal !!!
      CLR   ;
      =     DB1485.DBX   26.2;

//CIP Program Selected
      A     #CIP;
      =     DB1485.DBX   27.1;

// Emergency Stop
      A     #EStopOK; //If needed add or replace with own SpI
      =     DB1485.DBX   27.0; //Emergency Stop OK


NETWORK
TITLE = read from other unit data



END_FUNCTION_BLOCK

FUNCTION_BLOCK FB 1489
TITLE =U048: Water Transfer Plant 8
AUTHOR : Woermann
FAMILY : BOTEC_F1
NAME : Sim
VERSION : 0.1


VAR_TEMP
  CIP : BOOL ;	//CIP active
  xTmp : BOOL ;	//Temporary BOOL (free for general use)
  iTmp : INT ;	//Temporary INT (free for general use)
  rTmp : REAL ;	//Temporary REAL (free for general use)
  UnitNo : INT ;	//Unit Number
END_VAR
BEGIN
NETWORK
TITLE =General

      SET   ;
// get unit number ----------------------------------------------------------
      L     DB1480.DBW    0;
      T     #UnitNo;

// CIP ----------------------------------------------------------------------
      L     DB1481.DBD   54;
      L     0;
      <D    ;
      =     #CIP;

NETWORK
TITLE =Actuator

      A     DB1481.DBX   17.3;
      =     DB2480.DBX  425.3;
      =     DB2480.DBX  505.3;
      =     DB2480.DBX  585.3;
      =     DB2480.DBX  665.3;

NETWORK
TITLE =Special Input

      A     DB1481.DBX   17.3;

NETWORK
TITLE =Counter

      A     DB1481.DBX   17.3;
      A     M    101.0;


      CLR   ;
NETWORK
TITLE =Analog Input

      A     DB1481.DBX   17.3;

NETWORK
TITLE =Universal Value

      A     DB1481.DBX   17.3;
//      =     "U048UnVD".unv001.Sim;
//      =     "U048UnVD".unv002.Sim;
//      =     "U048UnVD".unv003.Sim;
//      =     "U048UnVD".unv004.Sim;

NETWORK
TITLE =PID

      A     DB1481.DBX   17.3;

NETWORK
TITLE =Message

      A     DB1481.DBX   17.3;
//      =     "U048MsgD".msg001.Sim;
//      =     "U048MsgD".msg002.Sim;
//      =     "U048MsgD".msg003.Sim;

NETWORK
TITLE =VLT

      A     DB1481.DBX   17.3;

END_FUNCTION_BLOCK

FUNCTION_BLOCK FB 1495
TITLE =U049: Water Transfer Plant 9
FAMILY : BOTEC_F1
NAME : Comm
VERSION : 0.1


VAR_TEMP
  iRetVal : INT ;	//return value as integer
  wRetVal : WORD ;	//return value as word
  Run : BOOL ;	//Unit in "RUN" mode
  EStopOK : BOOL ;	//Emergency Stop OK
  CIP : BOOL ;	//CIP Program Selected
  ComCIP : BOOL ;	//Communication with CIP Active
  xTmp : BOOL ;	//Temporary BOOL (free for general use)
  iTmp : INT ;	//Temporary INT (free for general use)
  rTmp : REAL ;	//Temporary REAL (free for general use)
  dTmp : DINT ;	//Temporary DINT (free for general use)
  UnitNo : INT ;	//Unit Number
  EquipmentID : INT ;	//Equipment ID
  Prid : DINT ;	//Process ID
  SFM36 : STRUCT 	// CIP Pump Mode
   I00 : BOOL ;	// Off
   I01 : BOOL ;	// Flow
   I02 : BOOL ;	// Pressure
   I03 : BOOL ;	// Fix Speed
   I04 : BOOL ;
   I05 : BOOL ;
   I06 : BOOL ;
   I07 : BOOL ;
   I08 : BOOL ;
   I09 : BOOL ;
   I10 : BOOL ;
   I11 : BOOL ;
   I12 : BOOL ;
   I13 : BOOL ;
   I14 : BOOL ;
   I15 : BOOL ;
   I16 : BOOL ;
   I17 : BOOL ;
   I18 : BOOL ;
   I19 : BOOL ;
   I20 : BOOL ;
   I21 : BOOL ;
   I22 : BOOL ;
   I23 : BOOL ;
   I24 : BOOL ;
   I25 : BOOL ;
   I26 : BOOL ;
   I27 : BOOL ;
   I28 : BOOL ;
   I29 : BOOL ;
   I30 : BOOL ;
   I31 : BOOL ;
  END_STRUCT ;
END_VAR
BEGIN
NETWORK
TITLE =general

      SET   ;

// unit & equipment number ---------------------------------------------------
      L     DB1490.DBW    0;
      T     #UnitNo;

      L     DB1495.DBW   14;
      L     1000;
      *I    ;
      L     #UnitNo;
      +I    ;
      T     #EquipmentID;

// CIP ----------------------------------------------------------------------
      L     DB1495.DBW   18;
      L     0;
      <I    ;
      =     #CIP;

// Communicating Units-------------------------------------------------------
      L     DB1495.DBD   10;
      L     DB1495.DBD  106;
      ==D   ;
      =     #ComCIP;

// emergency OK -------------------------------------------------------------
      A     DB1495.DBX   75.0; //General Emergency Stop OK
      =     #EStopOK;

NETWORK
TITLE =read other unit's data

      SET   ;

// ... General Unit ----------/

      CALL FC   563 (
           ActReq                   := M    101.0,
           PLCNo                    := DB1495.DBW   14,
           SourceUnitNo             := 99,
           IsTUnit                  := FALSE,
           DstComDRec               := DB1495.GEN,
           RET_VAL                  := #wRetVal);

NETWORK
TITLE =remote start

      SET   ;
// !!! insert correct condition of unit start !!!
      A     DB1491.DBX   15.0;
      A     DB1491.DBX   17.4;
      CLR   ;
      JCN   Strt;
      L     DB1495.DBD   10;
//L        L#-1;                            // Prid negative to start on its own
      T     #Prid;

      CALL FC    48 (
           UnitNo                   := #UnitNo,
           PrId                     := #Prid,
           Run                      := DB1491.DBX   17.4,
           PrIdTransfer             := TRUE,
           Start                    := TRUE,
           RetVal                   := #wRetVal);
Strt: NOP   0;
NETWORK
TITLE =external releases

      SET   ;
      =     DB2490.DBX  186.7;
      =     DB2490.DBX  266.7;
      =     DB2490.DBX  346.7;
      =     DB2490.DBX  426.7;
      =     DB2490.DBX  506.7;
      =     DB2490.DBX  586.7;
      =     DB2490.DBX  666.7;
NETWORK
TITLE =write own unit data

      SET   ;

//-- CIP Communication ---------------------------------------
      AN    DB1491.DBX   15.0;
//      AN "U049SeqD".Seq.PO.B30 // CIP Active (Slave)
      A     #ComCIP;
      JCN   NCIP;
//Conductivity CIP Return
      L     DB1495.DBD  150;
      T     DB1491.DBD  626;

//Temperature CIP Return
      L     DB1495.DBD  146;
      T     DB1491.DBD  594;

//CIP Prerun Pump SP

      CALL FC    45 (
           SFM                      := DB1491.DBD  686,
           Indexes                  := #SFM36);


      L     0.000000e+000;
      A     #SFM36.I01;
      =     DB1495.DBX  171.7;
      JCN   pfc;
      L     DB1491.DBD  654;
pfc:  NOP   0;
      A     #SFM36.I02;
      =     DB1495.DBX  172.0;
      JCN   ppc;
      L     DB1491.DBD  670;
ppc:  NOP   0;
      A     #SFM36.I03;
      =     DB1495.DBX  171.6;
      JCN   pxc;
      L     DB1491.DBD  574;
pxc:  NOP   0;
      T     DB1495.DBD  182;

//CIP Return
      L     DB1491.DBD  558;
      T     DB1495.DBD  186;
      L     DB1495.DBD  138;
      T     DB1491.DBD  562;

//CIP Prerun
      L     DB1491.DBD  542;
      T     DB1495.DBD  190;
      L     DB1495.DBD  142;
      T     DB1491.DBD  546;

// Write Own Data to CIP
      L     DB1495.DBD   10;
      T     DB1495.DBD  154;

      L     DB1495.DBW   14;
      T     DB1495.DBW  158;

      L     DB1495.DBW   16;
      T     DB1495.DBW  160;

      L     DB1495.DBW   18;
      T     DB1495.DBW  162;

      L     DB1495.DBW   20;
      T     DB1495.DBW  164;

      L     DB1495.DBW   22;
      T     DB1495.DBW  166;

      A     DB1495.DBX   24.0;
      =     DB1495.DBX  168.0;

      A     DB1495.DBX   24.1;
      =     DB1495.DBX  168.1;

      A     DB1495.DBX   24.2;
      =     DB1495.DBX  168.2;

      A     DB1495.DBX   24.3;
      =     DB1495.DBX  168.3;

      A     DB1495.DBX   24.4;
      =     DB1495.DBX  168.4;

      A     DB1495.DBX   24.5;
      =     DB1495.DBX  168.5;

      A     DB1495.DBX   24.6;
      =     DB1495.DBX  168.6;

      A     DB1495.DBX   24.7;
      =     DB1495.DBX  168.7;

// Copy Data to CIP
      CALL SFC   20 (
           SRCBLK                   := DB1495.ToCIP,
           RET_VAL                  := #iRetVal,
           DSTBLK                   := DB1495.ToCIP);

NCIP: NOP   0;

//Empty Signal
//A     "U049SpID".SpI.Sig //!!!! Insert correct Empty Signal !!!
      CLR   ;
      =     DB1495.DBX   26.5;

//Full Signal
//A     "U049SpID".SpI.Sig //!!!! Insert correct Full Signal !!!
      CLR   ;
      =     DB1495.DBX   26.2;

//CIP Program Selected
      A     #CIP;
      =     DB1495.DBX   27.1;

// Emergency Stop
      A     #EStopOK; //If needed add or replace with own SpI
      =     DB1495.DBX   27.0; //Emergency Stop OK


NETWORK
TITLE = read from other unit data



END_FUNCTION_BLOCK

FUNCTION_BLOCK FB 1499
TITLE =U049: Water Transfer Plant 9
AUTHOR : Woermann
FAMILY : BOTEC_F1
NAME : Sim
VERSION : 0.1


VAR_TEMP
  CIP : BOOL ;	//CIP active
  xTmp : BOOL ;	//Temporary BOOL (free for general use)
  iTmp : INT ;	//Temporary INT (free for general use)
  rTmp : REAL ;	//Temporary REAL (free for general use)
  UnitNo : INT ;	//Unit Number
END_VAR
BEGIN
NETWORK
TITLE =General

      SET   ;
// get unit number ----------------------------------------------------------
      L     DB1490.DBW    0;
      T     #UnitNo;

// CIP ----------------------------------------------------------------------
      L     DB1491.DBD   54;
      L     0;
      <D    ;
      =     #CIP;

NETWORK
TITLE =Actuator

      A     DB1491.DBX   17.3;
      =     DB2490.DBX  185.3;
      =     DB2490.DBX  265.3;
      =     DB2490.DBX  345.3;
      =     DB2490.DBX  425.3;
      =     DB2490.DBX  505.3;
      =     DB2490.DBX  585.3;
      =     DB2490.DBX  665.3;

NETWORK
TITLE =Special Input

      A     DB1491.DBX   17.3;

NETWORK
TITLE =Counter

      A     DB1491.DBX   17.3;
      A     M    101.0;


      CLR   ;
NETWORK
TITLE =Analog Input

      A     DB1491.DBX   17.3;

NETWORK
TITLE =Universal Value

      A     DB1491.DBX   17.3;
//      =     "U049UnVD".unv001.Sim;
//      =     "U049UnVD".unv002.Sim;
//      =     "U049UnVD".unv003.Sim;
//      =     "U049UnVD".unv004.Sim;

NETWORK
TITLE =PID

      A     DB1491.DBX   17.3;

NETWORK
TITLE =Message

      A     DB1491.DBX   17.3;
//      =     "U049MsgD".msg001.Sim;
//      =     "U049MsgD".msg002.Sim;
//      =     "U049MsgD".msg003.Sim;

NETWORK
TITLE =VLT

      A     DB1491.DBX   17.3;

END_FUNCTION_BLOCK

FUNCTION_BLOCK FB 1505
TITLE =U050: Water Transfer Plant 10
FAMILY : BOTEC_F1
NAME : Comm
VERSION : 0.1


VAR_TEMP
  iRetVal : INT ;	//return value as integer
  wRetVal : WORD ;	//return value as word
  Run : BOOL ;	//Unit in "RUN" mode
  EStopOK : BOOL ;	//Emergency Stop OK
  CIP : BOOL ;	//CIP Program Selected
  ComCIP : BOOL ;	//Communication with CIP Active
  xTmp : BOOL ;	//Temporary BOOL (free for general use)
  iTmp : INT ;	//Temporary INT (free for general use)
  rTmp : REAL ;	//Temporary REAL (free for general use)
  dTmp : DINT ;	//Temporary DINT (free for general use)
  UnitNo : INT ;	//Unit Number
  EquipmentID : INT ;	//Equipment ID
  Prid : DINT ;	//Process ID
  SFM36 : STRUCT 	// CIP Pump Mode
   I00 : BOOL ;	// Off
   I01 : BOOL ;	// Flow
   I02 : BOOL ;	// Pressure
   I03 : BOOL ;	// Fix Speed
   I04 : BOOL ;
   I05 : BOOL ;
   I06 : BOOL ;
   I07 : BOOL ;
   I08 : BOOL ;
   I09 : BOOL ;
   I10 : BOOL ;
   I11 : BOOL ;
   I12 : BOOL ;
   I13 : BOOL ;
   I14 : BOOL ;
   I15 : BOOL ;
   I16 : BOOL ;
   I17 : BOOL ;
   I18 : BOOL ;
   I19 : BOOL ;
   I20 : BOOL ;
   I21 : BOOL ;
   I22 : BOOL ;
   I23 : BOOL ;
   I24 : BOOL ;
   I25 : BOOL ;
   I26 : BOOL ;
   I27 : BOOL ;
   I28 : BOOL ;
   I29 : BOOL ;
   I30 : BOOL ;
   I31 : BOOL ;
  END_STRUCT ;
END_VAR
BEGIN
NETWORK
TITLE =general

      SET   ;

// unit & equipment number ---------------------------------------------------
      L     DB1500.DBW    0;
      T     #UnitNo;

      L     DB1505.DBW   14;
      L     1000;
      *I    ;
      L     #UnitNo;
      +I    ;
      T     #EquipmentID;

// CIP ----------------------------------------------------------------------
      L     DB1505.DBW   18;
      L     0;
      <I    ;
      =     #CIP;

// Communicating Units-------------------------------------------------------
      L     DB1505.DBD   10;
      L     DB1505.DBD  106;
      ==D   ;
      =     #ComCIP;

// emergency OK -------------------------------------------------------------
      A     DB1505.DBX   75.0; //General Emergency Stop OK
      =     #EStopOK;

NETWORK
TITLE =read other unit's data

      SET   ;

// ... General Unit ----------/

      CALL FC   563 (
           ActReq                   := M    101.0,
           PLCNo                    := DB1505.DBW   14,
           SourceUnitNo             := 99,
           IsTUnit                  := FALSE,
           DstComDRec               := DB1505.GEN,
           RET_VAL                  := #wRetVal);

NETWORK
TITLE =remote start

      SET   ;
// !!! insert correct condition of unit start !!!
      A     DB1501.DBX   15.0;
      A     DB1501.DBX   17.4;
      CLR   ;
      JCN   Strt;
      L     DB1505.DBD   10;
//L        L#-1;                            // Prid negative to start on its own
      T     #Prid;

      CALL FC    48 (
           UnitNo                   := #UnitNo,
           PrId                     := #Prid,
           Run                      := DB1501.DBX   17.4,
           PrIdTransfer             := TRUE,
           Start                    := TRUE,
           RetVal                   := #wRetVal);
Strt: NOP   0;
NETWORK
TITLE =external releases

      SET   ;
      =     DB2500.DBX  186.7;
      =     DB2500.DBX  266.7;
      =     DB2500.DBX  346.7;
      =     DB2500.DBX  426.7;
      =     DB2500.DBX  506.7;
      =     DB2500.DBX  586.7;
      =     DB2500.DBX  666.7;
NETWORK
TITLE =write own unit data

      SET   ;

//-- CIP Communication ---------------------------------------
      AN    DB1501.DBX   15.0;
//      AN "U050SeqD".Seq.PO.B30 // CIP Active (Slave)
      A     #ComCIP;
      JCN   NCIP;
//Conductivity CIP Return
      L     DB1505.DBD  150;
      T     DB1501.DBD  626;

//Temperature CIP Return
      L     DB1505.DBD  146;
      T     DB1501.DBD  594;

//CIP Prerun Pump SP

      CALL FC    45 (
           SFM                      := DB1501.DBD  686,
           Indexes                  := #SFM36);


      L     0.000000e+000;
      A     #SFM36.I01;
      =     DB1505.DBX  171.7;
      JCN   pfc;
      L     DB1501.DBD  654;
pfc:  NOP   0;
      A     #SFM36.I02;
      =     DB1505.DBX  172.0;
      JCN   ppc;
      L     DB1501.DBD  670;
ppc:  NOP   0;
      A     #SFM36.I03;
      =     DB1505.DBX  171.6;
      JCN   pxc;
      L     DB1501.DBD  574;
pxc:  NOP   0;
      T     DB1505.DBD  182;

//CIP Return
      L     DB1501.DBD  558;
      T     DB1505.DBD  186;
      L     DB1505.DBD  138;
      T     DB1501.DBD  562;

//CIP Prerun
      L     DB1501.DBD  542;
      T     DB1505.DBD  190;
      L     DB1505.DBD  142;
      T     DB1501.DBD  546;

// Write Own Data to CIP
      L     DB1505.DBD   10;
      T     DB1505.DBD  154;

      L     DB1505.DBW   14;
      T     DB1505.DBW  158;

      L     DB1505.DBW   16;
      T     DB1505.DBW  160;

      L     DB1505.DBW   18;
      T     DB1505.DBW  162;

      L     DB1505.DBW   20;
      T     DB1505.DBW  164;

      L     DB1505.DBW   22;
      T     DB1505.DBW  166;

      A     DB1505.DBX   24.0;
      =     DB1505.DBX  168.0;

      A     DB1505.DBX   24.1;
      =     DB1505.DBX  168.1;

      A     DB1505.DBX   24.2;
      =     DB1505.DBX  168.2;

      A     DB1505.DBX   24.3;
      =     DB1505.DBX  168.3;

      A     DB1505.DBX   24.4;
      =     DB1505.DBX  168.4;

      A     DB1505.DBX   24.5;
      =     DB1505.DBX  168.5;

      A     DB1505.DBX   24.6;
      =     DB1505.DBX  168.6;

      A     DB1505.DBX   24.7;
      =     DB1505.DBX  168.7;

// Copy Data to CIP
      CALL SFC   20 (
           SRCBLK                   := DB1505.ToCIP,
           RET_VAL                  := #iRetVal,
           DSTBLK                   := DB1505.ToCIP);

NCIP: NOP   0;

//Empty Signal
//A     "U050SpID".SpI.Sig //!!!! Insert correct Empty Signal !!!
      CLR   ;
      =     DB1505.DBX   26.5;

//Full Signal
//A     "U050SpID".SpI.Sig //!!!! Insert correct Full Signal !!!
      CLR   ;
      =     DB1505.DBX   26.2;

//CIP Program Selected
      A     #CIP;
      =     DB1505.DBX   27.1;

// Emergency Stop
      A     #EStopOK; //If needed add or replace with own SpI
      =     DB1505.DBX   27.0; //Emergency Stop OK


NETWORK
TITLE = read from other unit data



END_FUNCTION_BLOCK

FUNCTION_BLOCK FB 1509
TITLE =U050: Water Transfer Plant 10
AUTHOR : Woermann
FAMILY : BOTEC_F1
NAME : Sim
VERSION : 0.1


VAR_TEMP
  CIP : BOOL ;	//CIP active
  xTmp : BOOL ;	//Temporary BOOL (free for general use)
  iTmp : INT ;	//Temporary INT (free for general use)
  rTmp : REAL ;	//Temporary REAL (free for general use)
  UnitNo : INT ;	//Unit Number
END_VAR
BEGIN
NETWORK
TITLE =General

      SET   ;
// get unit number ----------------------------------------------------------
      L     DB1500.DBW    0;
      T     #UnitNo;

// CIP ----------------------------------------------------------------------
      L     DB1501.DBD   54;
      L     0;
      <D    ;
      =     #CIP;

NETWORK
TITLE =Actuator

      A     DB1501.DBX   17.3;
      =     DB2500.DBX  185.3;
      =     DB2500.DBX  265.3;
      =     DB2500.DBX  345.3;
      =     DB2500.DBX  425.3;
      =     DB2500.DBX  505.3;
      =     DB2500.DBX  585.3;
      =     DB2500.DBX  665.3;

NETWORK
TITLE =Special Input

      A     DB1501.DBX   17.3;

NETWORK
TITLE =Counter

      A     DB1501.DBX   17.3;
      A     M    101.0;


      CLR   ;
NETWORK
TITLE =Analog Input

      A     DB1501.DBX   17.3;

NETWORK
TITLE =Universal Value

      A     DB1501.DBX   17.3;
//      =     "U050UnVD".unv001.Sim;
//      =     "U050UnVD".unv002.Sim;
//      =     "U050UnVD".unv003.Sim;
//      =     "U050UnVD".unv004.Sim;

NETWORK
TITLE =PID

      A     DB1501.DBX   17.3;

NETWORK
TITLE =Message

      A     DB1501.DBX   17.3;
//      =     "U050MsgD".msg001.Sim;
//      =     "U050MsgD".msg002.Sim;
//      =     "U050MsgD".msg003.Sim;

NETWORK
TITLE =VLT

      A     DB1501.DBX   17.3;

END_FUNCTION_BLOCK

FUNCTION_BLOCK FB 1515
TITLE =U051: Water Transfer Plant 11
FAMILY : BOTEC_F1
NAME : Comm
VERSION : 0.1


VAR_TEMP
  iRetVal : INT ;	//return value as integer
  wRetVal : WORD ;	//return value as word
  Run : BOOL ;	//Unit in "RUN" mode
  EStopOK : BOOL ;	//Emergency Stop OK
  CIP : BOOL ;	//CIP Program Selected
  ComCIP : BOOL ;	//Communication with CIP Active
  xTmp : BOOL ;	//Temporary BOOL (free for general use)
  iTmp : INT ;	//Temporary INT (free for general use)
  rTmp : REAL ;	//Temporary REAL (free for general use)
  dTmp : DINT ;	//Temporary DINT (free for general use)
  UnitNo : INT ;	//Unit Number
  EquipmentID : INT ;	//Equipment ID
  Prid : DINT ;	//Process ID
  SFM36 : STRUCT 	// CIP Pump Mode
   I00 : BOOL ;	// Off
   I01 : BOOL ;	// Flow
   I02 : BOOL ;	// Pressure
   I03 : BOOL ;	// Fix Speed
   I04 : BOOL ;
   I05 : BOOL ;
   I06 : BOOL ;
   I07 : BOOL ;
   I08 : BOOL ;
   I09 : BOOL ;
   I10 : BOOL ;
   I11 : BOOL ;
   I12 : BOOL ;
   I13 : BOOL ;
   I14 : BOOL ;
   I15 : BOOL ;
   I16 : BOOL ;
   I17 : BOOL ;
   I18 : BOOL ;
   I19 : BOOL ;
   I20 : BOOL ;
   I21 : BOOL ;
   I22 : BOOL ;
   I23 : BOOL ;
   I24 : BOOL ;
   I25 : BOOL ;
   I26 : BOOL ;
   I27 : BOOL ;
   I28 : BOOL ;
   I29 : BOOL ;
   I30 : BOOL ;
   I31 : BOOL ;
  END_STRUCT ;
END_VAR
BEGIN
NETWORK
TITLE =general

      SET   ;

// unit & equipment number ---------------------------------------------------
      L     DB1510.DBW    0;
      T     #UnitNo;

      L     DB1515.DBW   14;
      L     1000;
      *I    ;
      L     #UnitNo;
      +I    ;
      T     #EquipmentID;

// CIP ----------------------------------------------------------------------
      L     DB1515.DBW   18;
      L     0;
      <I    ;
      =     #CIP;

// Communicating Units-------------------------------------------------------
      L     DB1515.DBD   10;
      L     DB1515.DBD  106;
      ==D   ;
      =     #ComCIP;

// emergency OK -------------------------------------------------------------
      A     DB1515.DBX   75.0; //General Emergency Stop OK
      =     #EStopOK;

NETWORK
TITLE =read other unit's data

      SET   ;

// ... General Unit ----------/

      CALL FC   563 (
           ActReq                   := M    101.0,
           PLCNo                    := DB1515.DBW   14,
           SourceUnitNo             := 99,
           IsTUnit                  := FALSE,
           DstComDRec               := DB1515.GEN,
           RET_VAL                  := #wRetVal);

NETWORK
TITLE =remote start

      SET   ;
// !!! insert correct condition of unit start !!!
      A     DB1511.DBX   15.0;
      A     DB1511.DBX   17.4;
      CLR   ;
      JCN   Strt;
      L     DB1515.DBD   10;
//L        L#-1;                            // Prid negative to start on its own
      T     #Prid;

      CALL FC    48 (
           UnitNo                   := #UnitNo,
           PrId                     := #Prid,
           Run                      := DB1511.DBX   17.4,
           PrIdTransfer             := TRUE,
           Start                    := TRUE,
           RetVal                   := #wRetVal);
Strt: NOP   0;
NETWORK
TITLE =external releases

      SET   ;
      =     DB2510.DBX  186.7;
      =     DB2510.DBX  266.7;
      =     DB2510.DBX  346.7;
      =     DB2510.DBX  426.7;
      =     DB2510.DBX  506.7;
      =     DB2510.DBX  586.7;
      =     DB2510.DBX  666.7;
      =     DB2510.DBX  746.7;
NETWORK
TITLE =write own unit data

      SET   ;

//-- CIP Communication ---------------------------------------
      AN    DB1511.DBX   15.0;
//      AN "U051SeqD".Seq.PO.B30 // CIP Active (Slave)
      A     #ComCIP;
      JCN   NCIP;
//Conductivity CIP Return
      L     DB1515.DBD  150;
      T     DB1511.DBD  626;

//Temperature CIP Return
      L     DB1515.DBD  146;
      T     DB1511.DBD  594;

//CIP Prerun Pump SP

      CALL FC    45 (
           SFM                      := DB1511.DBD  686,
           Indexes                  := #SFM36);


      L     0.000000e+000;
      A     #SFM36.I01;
      =     DB1515.DBX  171.7;
      JCN   pfc;
      L     DB1511.DBD  654;
pfc:  NOP   0;
      A     #SFM36.I02;
      =     DB1515.DBX  172.0;
      JCN   ppc;
      L     DB1511.DBD  670;
ppc:  NOP   0;
      A     #SFM36.I03;
      =     DB1515.DBX  171.6;
      JCN   pxc;
      L     DB1511.DBD  574;
pxc:  NOP   0;
      T     DB1515.DBD  182;

//CIP Return
      L     DB1511.DBD  558;
      T     DB1515.DBD  186;
      L     DB1515.DBD  138;
      T     DB1511.DBD  562;

//CIP Prerun
      L     DB1511.DBD  542;
      T     DB1515.DBD  190;
      L     DB1515.DBD  142;
      T     DB1511.DBD  546;

// Write Own Data to CIP
      L     DB1515.DBD   10;
      T     DB1515.DBD  154;

      L     DB1515.DBW   14;
      T     DB1515.DBW  158;

      L     DB1515.DBW   16;
      T     DB1515.DBW  160;

      L     DB1515.DBW   18;
      T     DB1515.DBW  162;

      L     DB1515.DBW   20;
      T     DB1515.DBW  164;

      L     DB1515.DBW   22;
      T     DB1515.DBW  166;

      A     DB1515.DBX   24.0;
      =     DB1515.DBX  168.0;

      A     DB1515.DBX   24.1;
      =     DB1515.DBX  168.1;

      A     DB1515.DBX   24.2;
      =     DB1515.DBX  168.2;

      A     DB1515.DBX   24.3;
      =     DB1515.DBX  168.3;

      A     DB1515.DBX   24.4;
      =     DB1515.DBX  168.4;

      A     DB1515.DBX   24.5;
      =     DB1515.DBX  168.5;

      A     DB1515.DBX   24.6;
      =     DB1515.DBX  168.6;

      A     DB1515.DBX   24.7;
      =     DB1515.DBX  168.7;

// Copy Data to CIP
      CALL SFC   20 (
           SRCBLK                   := DB1515.ToCIP,
           RET_VAL                  := #iRetVal,
           DSTBLK                   := DB1515.ToCIP);

NCIP: NOP   0;

//Empty Signal
//A     "U051SpID".SpI.Sig //!!!! Insert correct Empty Signal !!!
      CLR   ;
      =     DB1515.DBX   26.5;

//Full Signal
//A     "U051SpID".SpI.Sig //!!!! Insert correct Full Signal !!!
      CLR   ;
      =     DB1515.DBX   26.2;

//CIP Program Selected
      A     #CIP;
      =     DB1515.DBX   27.1;

// Emergency Stop
      A     #EStopOK; //If needed add or replace with own SpI
      =     DB1515.DBX   27.0; //Emergency Stop OK


NETWORK
TITLE = read from other unit data



END_FUNCTION_BLOCK

FUNCTION_BLOCK FB 1519
TITLE =U051: Water Transfer Plant 11
AUTHOR : Woermann
FAMILY : BOTEC_F1
NAME : Sim
VERSION : 0.1


VAR_TEMP
  CIP : BOOL ;	//CIP active
  xTmp : BOOL ;	//Temporary BOOL (free for general use)
  iTmp : INT ;	//Temporary INT (free for general use)
  rTmp : REAL ;	//Temporary REAL (free for general use)
  UnitNo : INT ;	//Unit Number
END_VAR
BEGIN
NETWORK
TITLE =General

      SET   ;
// get unit number ----------------------------------------------------------
      L     DB1510.DBW    0;
      T     #UnitNo;

// CIP ----------------------------------------------------------------------
      L     DB1511.DBD   54;
      L     0;
      <D    ;
      =     #CIP;

NETWORK
TITLE =Actuator

      A     DB1511.DBX   17.3;
      =     DB2510.DBX  185.3;
      =     DB2510.DBX  265.3;
      =     DB2510.DBX  345.3;
      =     DB2510.DBX  425.3;
      =     DB2510.DBX  505.3;
      =     DB2510.DBX  585.3;
      =     DB2510.DBX  665.3;
      =     DB2510.DBX  745.3;

NETWORK
TITLE =Special Input

      A     DB1511.DBX   17.3;

NETWORK
TITLE =Counter

      A     DB1511.DBX   17.3;
      A     M    101.0;


      CLR   ;
NETWORK
TITLE =Analog Input

      A     DB1511.DBX   17.3;

NETWORK
TITLE =Universal Value

      A     DB1511.DBX   17.3;
//      =     "U051UnVD".unv001.Sim;
//      =     "U051UnVD".unv002.Sim;
//      =     "U051UnVD".unv003.Sim;
//      =     "U051UnVD".unv004.Sim;

NETWORK
TITLE =PID

      A     DB1511.DBX   17.3;

NETWORK
TITLE =Message

      A     DB1511.DBX   17.3;
//      =     "U051MsgD".msg001.Sim;
//      =     "U051MsgD".msg002.Sim;
//      =     "U051MsgD".msg003.Sim;

NETWORK
TITLE =VLT

      A     DB1511.DBX   17.3;

END_FUNCTION_BLOCK

FUNCTION_BLOCK FB 1525
TITLE =U052: Water Transfer Plant 12
FAMILY : BOTEC_F1
NAME : Comm
VERSION : 0.1


VAR_TEMP
  iRetVal : INT ;	//return value as integer
  wRetVal : WORD ;	//return value as word
  Run : BOOL ;	//Unit in "RUN" mode
  EStopOK : BOOL ;	//Emergency Stop OK
  CIP : BOOL ;	//CIP Program Selected
  ComCIP : BOOL ;	//Communication with CIP Active
  xTmp : BOOL ;	//Temporary BOOL (free for general use)
  iTmp : INT ;	//Temporary INT (free for general use)
  rTmp : REAL ;	//Temporary REAL (free for general use)
  dTmp : DINT ;	//Temporary DINT (free for general use)
  UnitNo : INT ;	//Unit Number
  EquipmentID : INT ;	//Equipment ID
  Prid : DINT ;	//Process ID
  SFM36 : STRUCT 	// CIP Pump Mode
   I00 : BOOL ;	// Off
   I01 : BOOL ;	// Flow
   I02 : BOOL ;	// Pressure
   I03 : BOOL ;	// Fix Speed
   I04 : BOOL ;
   I05 : BOOL ;
   I06 : BOOL ;
   I07 : BOOL ;
   I08 : BOOL ;
   I09 : BOOL ;
   I10 : BOOL ;
   I11 : BOOL ;
   I12 : BOOL ;
   I13 : BOOL ;
   I14 : BOOL ;
   I15 : BOOL ;
   I16 : BOOL ;
   I17 : BOOL ;
   I18 : BOOL ;
   I19 : BOOL ;
   I20 : BOOL ;
   I21 : BOOL ;
   I22 : BOOL ;
   I23 : BOOL ;
   I24 : BOOL ;
   I25 : BOOL ;
   I26 : BOOL ;
   I27 : BOOL ;
   I28 : BOOL ;
   I29 : BOOL ;
   I30 : BOOL ;
   I31 : BOOL ;
  END_STRUCT ;
END_VAR
BEGIN
NETWORK
TITLE =general

      SET   ;

// unit & equipment number ---------------------------------------------------
      L     DB1520.DBW    0;
      T     #UnitNo;

      L     DB1525.DBW   14;
      L     1000;
      *I    ;
      L     #UnitNo;
      +I    ;
      T     #EquipmentID;

// CIP ----------------------------------------------------------------------
      L     DB1525.DBW   18;
      L     0;
      <I    ;
      =     #CIP;

// Communicating Units-------------------------------------------------------
      L     DB1525.DBD   10;
      L     DB1525.DBD  106;
      ==D   ;
      =     #ComCIP;

// emergency OK -------------------------------------------------------------
      A     DB1525.DBX   75.0; //General Emergency Stop OK
      =     #EStopOK;

NETWORK
TITLE =read other unit's data

      SET   ;

// ... General Unit ----------/

      CALL FC   563 (
           ActReq                   := M    101.0,
           PLCNo                    := DB1525.DBW   14,
           SourceUnitNo             := 99,
           IsTUnit                  := FALSE,
           DstComDRec               := DB1525.GEN,
           RET_VAL                  := #wRetVal);


NETWORK
TITLE =remote start

      SET   ;
// !!! insert correct condition of unit start !!!
      A     DB1521.DBX   15.0;
      A     DB1521.DBX   17.4;
      CLR   ;
      JCN   Strt;
      L     DB1525.DBD   10;
//L        L#-1;                            // Prid negative to start on its own
      T     #Prid;

      CALL FC    48 (
           UnitNo                   := #UnitNo,
           PrId                     := #Prid,
           Run                      := DB1521.DBX   17.4,
           PrIdTransfer             := TRUE,
           Start                    := TRUE,
           RetVal                   := #wRetVal);
Strt: NOP   0;
NETWORK
TITLE =external releases

      SET   ;
      =     DB2520.DBX  186.7;
      =     DB2520.DBX  266.7;
      =     DB2520.DBX  346.7;
      =     DB2520.DBX  426.7;
      =     DB2520.DBX  506.7;
      =     DB2520.DBX  586.7;
      =     DB2520.DBX  666.7;
NETWORK
TITLE =write own unit data

      SET   ;

//-- CIP Communication ---------------------------------------
      AN    DB1521.DBX   15.0;
//      AN "U052SeqD".Seq.PO.B30 // CIP Active (Slave)
      A     #ComCIP;
      JCN   NCIP;
//Conductivity CIP Return
      L     DB1525.DBD  150;
      T     DB1521.DBD  626;

//Temperature CIP Return
      L     DB1525.DBD  146;
      T     DB1521.DBD  594;

//CIP Prerun Pump SP

      CALL FC    45 (
           SFM                      := DB1521.DBD  686,
           Indexes                  := #SFM36);


      L     0.000000e+000;
      A     #SFM36.I01;
      =     DB1525.DBX  171.7;
      JCN   pfc;
      L     DB1521.DBD  654;
pfc:  NOP   0;
      A     #SFM36.I02;
      =     DB1525.DBX  172.0;
      JCN   ppc;
      L     DB1521.DBD  670;
ppc:  NOP   0;
      A     #SFM36.I03;
      =     DB1525.DBX  171.6;
      JCN   pxc;
      L     DB1521.DBD  574;
pxc:  NOP   0;
      T     DB1525.DBD  182;

//CIP Return
      L     DB1521.DBD  558;
      T     DB1525.DBD  186;
      L     DB1525.DBD  138;
      T     DB1521.DBD  562;

//CIP Prerun
      L     DB1521.DBD  542;
      T     DB1525.DBD  190;
      L     DB1525.DBD  142;
      T     DB1521.DBD  546;

// Write Own Data to CIP
      L     DB1525.DBD   10;
      T     DB1525.DBD  154;

      L     DB1525.DBW   14;
      T     DB1525.DBW  158;

      L     DB1525.DBW   16;
      T     DB1525.DBW  160;

      L     DB1525.DBW   18;
      T     DB1525.DBW  162;

      L     DB1525.DBW   20;
      T     DB1525.DBW  164;

      L     DB1525.DBW   22;
      T     DB1525.DBW  166;

      A     DB1525.DBX   24.0;
      =     DB1525.DBX  168.0;

      A     DB1525.DBX   24.1;
      =     DB1525.DBX  168.1;

      A     DB1525.DBX   24.2;
      =     DB1525.DBX  168.2;

      A     DB1525.DBX   24.3;
      =     DB1525.DBX  168.3;

      A     DB1525.DBX   24.4;
      =     DB1525.DBX  168.4;

      A     DB1525.DBX   24.5;
      =     DB1525.DBX  168.5;

      A     DB1525.DBX   24.6;
      =     DB1525.DBX  168.6;

      A     DB1525.DBX   24.7;
      =     DB1525.DBX  168.7;

// Copy Data to CIP
      CALL SFC   20 (
           SRCBLK                   := DB1525.ToCIP,
           RET_VAL                  := #iRetVal,
           DSTBLK                   := DB1525.ToCIP);

NCIP: NOP   0;

//Empty Signal
//A     "U052SpID".SpI.Sig //!!!! Insert correct Empty Signal !!!
      CLR   ;
      =     DB1525.DBX   26.5;

//Full Signal
//A     "U052SpID".SpI.Sig //!!!! Insert correct Full Signal !!!
      CLR   ;
      =     DB1525.DBX   26.2;

//CIP Program Selected
      A     #CIP;
      =     DB1525.DBX   27.1;

// Emergency Stop
      A     #EStopOK; //If needed add or replace with own SpI
      =     DB1525.DBX   27.0; //Emergency Stop OK


NETWORK
TITLE = read from other unit data



END_FUNCTION_BLOCK

FUNCTION_BLOCK FB 1529
TITLE =U052: Water Transfer Plant 12
AUTHOR : Woermann
FAMILY : BOTEC_F1
NAME : Sim
VERSION : 0.1


VAR_TEMP
  CIP : BOOL ;	//CIP active
  xTmp : BOOL ;	//Temporary BOOL (free for general use)
  iTmp : INT ;	//Temporary INT (free for general use)
  rTmp : REAL ;	//Temporary REAL (free for general use)
  UnitNo : INT ;	//Unit Number
END_VAR
BEGIN
NETWORK
TITLE =General

      SET   ;
// get unit number ----------------------------------------------------------
      L     DB1520.DBW    0;
      T     #UnitNo;

// CIP ----------------------------------------------------------------------
      L     DB1521.DBD   54;
      L     0;
      <D    ;
      =     #CIP;

NETWORK
TITLE =Actuator

      A     DB1521.DBX   17.3;
      =     DB2520.DBX  185.3;
      =     DB2520.DBX  265.3;
      =     DB2520.DBX  345.3;
      =     DB2520.DBX  425.3;
      =     DB2520.DBX  505.3;
      =     DB2520.DBX  585.3;
      =     DB2520.DBX  665.3;

NETWORK
TITLE =Special Input

      A     DB1521.DBX   17.3;

NETWORK
TITLE =Counter

      A     DB1521.DBX   17.3;
      A     M    101.0;


      CLR   ;
NETWORK
TITLE =Analog Input

      A     DB1521.DBX   17.3;

NETWORK
TITLE =Universal Value

      A     DB1521.DBX   17.3;
//      =     "U052UnVD".unv001.Sim;
//      =     "U052UnVD".unv002.Sim;
//      =     "U052UnVD".unv003.Sim;
//      =     "U052UnVD".unv004.Sim;

NETWORK
TITLE =PID

      A     DB1521.DBX   17.3;

NETWORK
TITLE =Message

      A     DB1521.DBX   17.3;
//      =     "U052MsgD".msg001.Sim;
//      =     "U052MsgD".msg002.Sim;
//      =     "U052MsgD".msg003.Sim;

NETWORK
TITLE =VLT

      A     DB1521.DBX   17.3;

END_FUNCTION_BLOCK

FUNCTION_BLOCK FB 1545
TITLE =U054: Water Transfer Plant 14
FAMILY : BOTEC_F1
NAME : Comm
VERSION : 0.1


VAR_TEMP
  iRetVal : INT ;	//return value as integer
  wRetVal : WORD ;	//return value as word
  Run : BOOL ;	//Unit in "RUN" mode
  EStopOK : BOOL ;	//Emergency Stop OK
  CIP : BOOL ;	//CIP Program Selected
  ComCIP : BOOL ;	//Communication with CIP Active
  xTmp : BOOL ;	//Temporary BOOL (free for general use)
  iTmp : INT ;	//Temporary INT (free for general use)
  rTmp : REAL ;	//Temporary REAL (free for general use)
  dTmp : DINT ;	//Temporary DINT (free for general use)
  UnitNo : INT ;	//Unit Number
  EquipmentID : INT ;	//Equipment ID
  Prid : DINT ;	//Process ID
  SFM36 : STRUCT 	// CIP Pump Mode
   I00 : BOOL ;	// Off
   I01 : BOOL ;	// Flow
   I02 : BOOL ;	// Pressure
   I03 : BOOL ;	// Fix Speed
   I04 : BOOL ;
   I05 : BOOL ;
   I06 : BOOL ;
   I07 : BOOL ;
   I08 : BOOL ;
   I09 : BOOL ;
   I10 : BOOL ;
   I11 : BOOL ;
   I12 : BOOL ;
   I13 : BOOL ;
   I14 : BOOL ;
   I15 : BOOL ;
   I16 : BOOL ;
   I17 : BOOL ;
   I18 : BOOL ;
   I19 : BOOL ;
   I20 : BOOL ;
   I21 : BOOL ;
   I22 : BOOL ;
   I23 : BOOL ;
   I24 : BOOL ;
   I25 : BOOL ;
   I26 : BOOL ;
   I27 : BOOL ;
   I28 : BOOL ;
   I29 : BOOL ;
   I30 : BOOL ;
   I31 : BOOL ;
  END_STRUCT ;
END_VAR
BEGIN
NETWORK
TITLE =general

      SET   ;

// unit & equipment number ---------------------------------------------------
      L     DB1540.DBW    0;
      T     #UnitNo;

      L     DB1545.DBW   14;
      L     1000;
      *I    ;
      L     #UnitNo;
      +I    ;
      T     #EquipmentID;

// CIP ----------------------------------------------------------------------
      L     DB1545.DBW   18;
      L     0;
      <I    ;
      =     #CIP;

// Communicating Units-------------------------------------------------------
      L     DB1545.DBD   10;
      L     DB1545.DBD  106;
      ==D   ;
      =     #ComCIP;

// emergency OK -------------------------------------------------------------
      A     DB1545.DBX   75.0; //General Emergency Stop OK
      =     #EStopOK;

NETWORK
TITLE =read other unit's data

      SET   ;

// ... General Unit ----------/

      CALL FC   563 (
           ActReq                   := M    101.0,
           PLCNo                    := DB1545.DBW   14,
           SourceUnitNo             := 99,
           IsTUnit                  := FALSE,
           DstComDRec               := DB1545.GEN,
           RET_VAL                  := #wRetVal);

NETWORK
TITLE =remote start

      SET   ;
// !!! insert correct condition of unit start !!!
      A     DB1541.DBX   15.0;
      A     DB1541.DBX   17.4;
      CLR   ;
      JCN   Strt;
      L     DB1545.DBD   10;
//L        L#-1;                            // Prid negative to start on its own
      T     #Prid;

      CALL FC    48 (
           UnitNo                   := #UnitNo,
           PrId                     := #Prid,
           Run                      := DB1541.DBX   17.4,
           PrIdTransfer             := TRUE,
           Start                    := TRUE,
           RetVal                   := #wRetVal);
Strt: NOP   0;
NETWORK
TITLE =external releases

      SET   ;
      =     DB2540.DBX  186.7;
      =     DB2540.DBX  266.7;
      =     DB2540.DBX  346.7;
      =     DB2540.DBX  426.7;
      =     DB2540.DBX  506.7;
      =     DB2540.DBX  586.7;
      =     DB2540.DBX  666.7;
      =     DB2540.DBX  746.7;
      =     DB2540.DBX  826.7;

NETWORK
TITLE =write own unit data

      SET   ;

//-- CIP Communication ---------------------------------------
      AN    DB1541.DBX   15.0;
//      AN "U054SeqD".Seq.PO.B30 // CIP Active (Slave)
      A     #ComCIP;
      JCN   NCIP;
//Conductivity CIP Return
      L     DB1545.DBD  150;
      T     DB1541.DBD  626;

//Temperature CIP Return
      L     DB1545.DBD  146;
      T     DB1541.DBD  594;

//CIP Prerun Pump SP

      CALL FC    45 (
           SFM                      := DB1541.DBD  686,
           Indexes                  := #SFM36);


      L     0.000000e+000;
      A     #SFM36.I01;
      =     DB1545.DBX  171.7;
      JCN   pfc;
      L     DB1541.DBD  654;
pfc:  NOP   0;
      A     #SFM36.I02;
      =     DB1545.DBX  172.0;
      JCN   ppc;
      L     DB1541.DBD  670;
ppc:  NOP   0;
      A     #SFM36.I03;
      =     DB1545.DBX  171.6;
      JCN   pxc;
      L     DB1541.DBD  574;
pxc:  NOP   0;
      T     DB1545.DBD  182;

//CIP Return
      L     DB1541.DBD  558;
      T     DB1545.DBD  186;
      L     DB1545.DBD  138;
      T     DB1541.DBD  562;

//CIP Prerun
      L     DB1541.DBD  542;
      T     DB1545.DBD  190;
      L     DB1545.DBD  142;
      T     DB1541.DBD  546;

// Write Own Data to CIP
      L     DB1545.DBD   10;
      T     DB1545.DBD  154;

      L     DB1545.DBW   14;
      T     DB1545.DBW  158;

      L     DB1545.DBW   16;
      T     DB1545.DBW  160;

      L     DB1545.DBW   18;
      T     DB1545.DBW  162;

      L     DB1545.DBW   20;
      T     DB1545.DBW  164;

      L     DB1545.DBW   22;
      T     DB1545.DBW  166;

      A     DB1545.DBX   24.0;
      =     DB1545.DBX  168.0;

      A     DB1545.DBX   24.1;
      =     DB1545.DBX  168.1;

      A     DB1545.DBX   24.2;
      =     DB1545.DBX  168.2;

      A     DB1545.DBX   24.3;
      =     DB1545.DBX  168.3;

      A     DB1545.DBX   24.4;
      =     DB1545.DBX  168.4;

      A     DB1545.DBX   24.5;
      =     DB1545.DBX  168.5;

      A     DB1545.DBX   24.6;
      =     DB1545.DBX  168.6;

      A     DB1545.DBX   24.7;
      =     DB1545.DBX  168.7;

// Copy Data to CIP
      CALL SFC   20 (
           SRCBLK                   := DB1545.ToCIP,
           RET_VAL                  := #iRetVal,
           DSTBLK                   := DB1545.ToCIP);

NCIP: NOP   0;

//Empty Signal
//A     "U054SpID".SpI.Sig //!!!! Insert correct Empty Signal !!!
      CLR   ;
      =     DB1545.DBX   26.5;

//Full Signal
//A     "U054SpID".SpI.Sig //!!!! Insert correct Full Signal !!!
      CLR   ;
      =     DB1545.DBX   26.2;

//CIP Program Selected
      A     #CIP;
      =     DB1545.DBX   27.1;

// Emergency Stop
      A     #EStopOK; //If needed add or replace with own SpI
      =     DB1545.DBX   27.0; //Emergency Stop OK


NETWORK
TITLE = read from other unit data



END_FUNCTION_BLOCK

FUNCTION_BLOCK FB 1549
TITLE =U054: Water Transfer Plant 14
AUTHOR : Woermann
FAMILY : BOTEC_F1
NAME : Sim
VERSION : 0.1


VAR_TEMP
  CIP : BOOL ;	//CIP active
  xTmp : BOOL ;	//Temporary BOOL (free for general use)
  iTmp : INT ;	//Temporary INT (free for general use)
  rTmp : REAL ;	//Temporary REAL (free for general use)
  UnitNo : INT ;	//Unit Number
END_VAR
BEGIN
NETWORK
TITLE =General

      SET   ;
// get unit number ----------------------------------------------------------
      L     DB1540.DBW    0;
      T     #UnitNo;

// CIP ----------------------------------------------------------------------
      L     DB1541.DBD   54;
      L     0;
      <D    ;
      =     #CIP;

NETWORK
TITLE =Actuator

      A     DB1541.DBX   17.3;
      =     DB2540.DBX  185.3;
      =     DB2540.DBX  265.3;
      =     DB2540.DBX  345.3;
      =     DB2540.DBX  425.3;
      =     DB2540.DBX  505.3;
      =     DB2540.DBX  585.3;
      =     DB2540.DBX  665.3;
      =     DB2540.DBX  745.3;
      =     DB2540.DBX  825.3;

NETWORK
TITLE =Special Input

      A     DB1541.DBX   17.3;

NETWORK
TITLE =Counter

      A     DB1541.DBX   17.3;
      A     M    101.0;


      CLR   ;
NETWORK
TITLE =Analog Input

      A     DB1541.DBX   17.3;

NETWORK
TITLE =Universal Value

      A     DB1541.DBX   17.3;
//      =     "U054UnVD".unv001.Sim;
//      =     "U054UnVD".unv002.Sim;
//      =     "U054UnVD".unv003.Sim;
//      =     "U054UnVD".unv004.Sim;

NETWORK
TITLE =PID

      A     DB1541.DBX   17.3;

NETWORK
TITLE =Message

      A     DB1541.DBX   17.3;
//      =     "U054MsgD".msg001.Sim;
//      =     "U054MsgD".msg002.Sim;
//      =     "U054MsgD".msg003.Sim;

NETWORK
TITLE =VLT

      A     DB1541.DBX   17.3;

END_FUNCTION_BLOCK

FUNCTION_BLOCK FB 1555
TITLE =U055: Water Transfer Plant 15
FAMILY : BOTEC_F1
NAME : Comm
VERSION : 0.1


VAR_TEMP
  iRetVal : INT ;	//return value as integer
  wRetVal : WORD ;	//return value as word
  Run : BOOL ;	//Unit in "RUN" mode
  EStopOK : BOOL ;	//Emergency Stop OK
  CIP : BOOL ;	//CIP Program Selected
  ComCIP : BOOL ;	//Communication with CIP Active
  xTmp : BOOL ;	//Temporary BOOL (free for general use)
  iTmp : INT ;	//Temporary INT (free for general use)
  rTmp : REAL ;	//Temporary REAL (free for general use)
  dTmp : DINT ;	//Temporary DINT (free for general use)
  UnitNo : INT ;	//Unit Number
  EquipmentID : INT ;	//Equipment ID
  Prid : DINT ;	//Process ID
  SFM36 : STRUCT 	// CIP Pump Mode
   I00 : BOOL ;	// Off
   I01 : BOOL ;	// Flow
   I02 : BOOL ;	// Pressure
   I03 : BOOL ;	// Fix Speed
   I04 : BOOL ;
   I05 : BOOL ;
   I06 : BOOL ;
   I07 : BOOL ;
   I08 : BOOL ;
   I09 : BOOL ;
   I10 : BOOL ;
   I11 : BOOL ;
   I12 : BOOL ;
   I13 : BOOL ;
   I14 : BOOL ;
   I15 : BOOL ;
   I16 : BOOL ;
   I17 : BOOL ;
   I18 : BOOL ;
   I19 : BOOL ;
   I20 : BOOL ;
   I21 : BOOL ;
   I22 : BOOL ;
   I23 : BOOL ;
   I24 : BOOL ;
   I25 : BOOL ;
   I26 : BOOL ;
   I27 : BOOL ;
   I28 : BOOL ;
   I29 : BOOL ;
   I30 : BOOL ;
   I31 : BOOL ;
  END_STRUCT ;
END_VAR
BEGIN
NETWORK
TITLE =general

      SET   ;

// unit & equipment number ---------------------------------------------------
      L     DB1550.DBW    0;
      T     #UnitNo;

      L     DB1555.DBW   14;
      L     1000;
      *I    ;
      L     #UnitNo;
      +I    ;
      T     #EquipmentID;

// CIP ----------------------------------------------------------------------
      L     DB1555.DBW   18;
      L     0;
      <I    ;
      =     #CIP;

// Communicating Units-------------------------------------------------------
      L     DB1555.DBD   10;
      L     DB1555.DBD  106;
      ==D   ;
      =     #ComCIP;

// emergency OK -------------------------------------------------------------
      A     DB1555.DBX   75.0; //General Emergency Stop OK
      =     #EStopOK;

NETWORK
TITLE =read other unit's data

      SET   ;

// ... General Unit ----------/

      CALL FC   563 (
           ActReq                   := M    101.0,
           PLCNo                    := DB1555.DBW   14,
           SourceUnitNo             := 99,
           IsTUnit                  := FALSE,
           DstComDRec               := DB1555.GEN,
           RET_VAL                  := #wRetVal);

NETWORK
TITLE =remote start

      SET   ;
// !!! insert correct condition of unit start !!!
      A     DB1551.DBX   15.0;
      A     DB1551.DBX   17.4;
      CLR   ;
      JCN   Strt;
      L     DB1555.DBD   10;
//L        L#-1;                            // Prid negative to start on its own
      T     #Prid;

      CALL FC    48 (
           UnitNo                   := #UnitNo,
           PrId                     := #Prid,
           Run                      := DB1551.DBX   17.4,
           PrIdTransfer             := TRUE,
           Start                    := TRUE,
           RetVal                   := #wRetVal);
Strt: NOP   0;
NETWORK
TITLE =external releases

      SET   ;
      =     DB2550.DBX  426.7;
      =     DB2550.DBX  506.7;
      =     DB2550.DBX  586.7;
NETWORK
TITLE =write own unit data

      SET   ;

//-- CIP Communication ---------------------------------------
      AN    DB1551.DBX   15.0;
//      AN "U055SeqD".Seq.PO.B30 // CIP Active (Slave)
      A     #ComCIP;
      JCN   NCIP;
//Conductivity CIP Return
      L     DB1555.DBD  150;
      T     DB1551.DBD  626;

//Temperature CIP Return
      L     DB1555.DBD  146;
      T     DB1551.DBD  594;

//CIP Prerun Pump SP

      CALL FC    45 (
           SFM                      := DB1551.DBD  686,
           Indexes                  := #SFM36);


      L     0.000000e+000;
      A     #SFM36.I01;
      =     DB1555.DBX  171.7;
      JCN   pfc;
      L     DB1551.DBD  654;
pfc:  NOP   0;
      A     #SFM36.I02;
      =     DB1555.DBX  172.0;
      JCN   ppc;
      L     DB1551.DBD  670;
ppc:  NOP   0;
      A     #SFM36.I03;
      =     DB1555.DBX  171.6;
      JCN   pxc;
      L     DB1551.DBD  574;
pxc:  NOP   0;
      T     DB1555.DBD  182;

//CIP Return
      L     DB1551.DBD  558;
      T     DB1555.DBD  186;
      L     DB1555.DBD  138;
      T     DB1551.DBD  562;

//CIP Prerun
      L     DB1551.DBD  542;
      T     DB1555.DBD  190;
      L     DB1555.DBD  142;
      T     DB1551.DBD  546;

// Write Own Data to CIP
      L     DB1555.DBD   10;
      T     DB1555.DBD  154;

      L     DB1555.DBW   14;
      T     DB1555.DBW  158;

      L     DB1555.DBW   16;
      T     DB1555.DBW  160;

      L     DB1555.DBW   18;
      T     DB1555.DBW  162;

      L     DB1555.DBW   20;
      T     DB1555.DBW  164;

      L     DB1555.DBW   22;
      T     DB1555.DBW  166;

      A     DB1555.DBX   24.0;
      =     DB1555.DBX  168.0;

      A     DB1555.DBX   24.1;
      =     DB1555.DBX  168.1;

      A     DB1555.DBX   24.2;
      =     DB1555.DBX  168.2;

      A     DB1555.DBX   24.3;
      =     DB1555.DBX  168.3;

      A     DB1555.DBX   24.4;
      =     DB1555.DBX  168.4;

      A     DB1555.DBX   24.5;
      =     DB1555.DBX  168.5;

      A     DB1555.DBX   24.6;
      =     DB1555.DBX  168.6;

      A     DB1555.DBX   24.7;
      =     DB1555.DBX  168.7;

// Copy Data to CIP
      CALL SFC   20 (
           SRCBLK                   := DB1555.ToCIP,
           RET_VAL                  := #iRetVal,
           DSTBLK                   := DB1555.ToCIP);

NCIP: NOP   0;

//Empty Signal
//A     "U055SpID".SpI.Sig //!!!! Insert correct Empty Signal !!!
      CLR   ;
      =     DB1555.DBX   26.5;

//Full Signal
//A     "U055SpID".SpI.Sig //!!!! Insert correct Full Signal !!!
      CLR   ;
      =     DB1555.DBX   26.2;

//CIP Program Selected
      A     #CIP;
      =     DB1555.DBX   27.1;

// Emergency Stop
      A     #EStopOK; //If needed add or replace with own SpI
      =     DB1555.DBX   27.0; //Emergency Stop OK


NETWORK
TITLE = read from other unit data



END_FUNCTION_BLOCK

FUNCTION_BLOCK FB 1559
TITLE =U055: Water Transfer Plant 15
AUTHOR : Woermann
FAMILY : BOTEC_F1
NAME : Sim
VERSION : 0.1


VAR_TEMP
  CIP : BOOL ;	//CIP active
  xTmp : BOOL ;	//Temporary BOOL (free for general use)
  iTmp : INT ;	//Temporary INT (free for general use)
  rTmp : REAL ;	//Temporary REAL (free for general use)
  UnitNo : INT ;	//Unit Number
END_VAR
BEGIN
NETWORK
TITLE =General

      SET   ;
// get unit number ----------------------------------------------------------
      L     DB1550.DBW    0;
      T     #UnitNo;

// CIP ----------------------------------------------------------------------
      L     DB1551.DBD   54;
      L     0;
      <D    ;
      =     #CIP;

NETWORK
TITLE =Actuator

      A     DB1551.DBX   17.3;
      =     DB2550.DBX  425.3;
      =     DB2550.DBX  505.3;
      =     DB2550.DBX  585.3;

NETWORK
TITLE =Special Input

      A     DB1551.DBX   17.3;

NETWORK
TITLE =Counter

      A     DB1551.DBX   17.3;
      A     M    101.0;


      CLR   ;
NETWORK
TITLE =Analog Input

      A     DB1551.DBX   17.3;

NETWORK
TITLE =Universal Value

      A     DB1551.DBX   17.3;
//      =     "U055UnVD".unv001.Sim;
//      =     "U055UnVD".unv002.Sim;
//      =     "U055UnVD".unv003.Sim;
//      =     "U055UnVD".unv004.Sim;

NETWORK
TITLE =PID

      A     DB1551.DBX   17.3;

NETWORK
TITLE =Message

      A     DB1551.DBX   17.3;
//      =     "U055MsgD".msg001.Sim;
//      =     "U055MsgD".msg002.Sim;
//      =     "U055MsgD".msg003.Sim;

NETWORK
TITLE =VLT

      A     DB1551.DBX   17.3;

END_FUNCTION_BLOCK

FUNCTION_BLOCK FB 1565
TITLE =U056: Fresh Water Transfer
FAMILY : BOTEC_F1
NAME : Comm
VERSION : 0.1


VAR_TEMP
  iRetVal : INT ;	//return value as integer
  wRetVal : WORD ;	//return value as word
  Run : BOOL ;	//Unit in "RUN" mode
  EStopOK : BOOL ;	//Emergency Stop OK
  CIP : BOOL ;	//CIP Program Selected
  ComCIP : BOOL ;	//Communication with CIP Active
  xTmp : BOOL ;	//Temporary BOOL (free for general use)
  iTmp : INT ;	//Temporary INT (free for general use)
  rTmp : REAL ;	//Temporary REAL (free for general use)
  dTmp : DINT ;	//Temporary DINT (free for general use)
  UnitNo : INT ;	//Unit Number
  EquipmentID : INT ;	//Equipment ID
  Prid : DINT ;	//Process ID
  SFM36 : STRUCT 	// CIP Pump Mode
   I00 : BOOL ;	// Off
   I01 : BOOL ;	// Flow
   I02 : BOOL ;	// Pressure
   I03 : BOOL ;	// Fix Speed
   I04 : BOOL ;
   I05 : BOOL ;
   I06 : BOOL ;
   I07 : BOOL ;
   I08 : BOOL ;
   I09 : BOOL ;
   I10 : BOOL ;
   I11 : BOOL ;
   I12 : BOOL ;
   I13 : BOOL ;
   I14 : BOOL ;
   I15 : BOOL ;
   I16 : BOOL ;
   I17 : BOOL ;
   I18 : BOOL ;
   I19 : BOOL ;
   I20 : BOOL ;
   I21 : BOOL ;
   I22 : BOOL ;
   I23 : BOOL ;
   I24 : BOOL ;
   I25 : BOOL ;
   I26 : BOOL ;
   I27 : BOOL ;
   I28 : BOOL ;
   I29 : BOOL ;
   I30 : BOOL ;
   I31 : BOOL ;
  END_STRUCT ;
  iPLC : INT ;
  iUnit : INT ;
END_VAR
BEGIN
NETWORK
TITLE =general

      SET   ;

// unit & equipment number ---------------------------------------------------
      L     DB1560.DBW    0;
      T     #UnitNo;

      L     DB1565.DBW   14;
      L     1000;
      *I    ;
      L     #UnitNo;
      +I    ;
      T     #EquipmentID;

// CIP ----------------------------------------------------------------------
      L     DB1565.DBW   18;
      L     0;
      <I    ;
      =     #CIP;

// Communicating Units-------------------------------------------------------
      L     DB1565.DBD   10;
      L     DB1565.DBD  106;
      ==D   ;
      =     #ComCIP;

// emergency OK -------------------------------------------------------------
      A     DB1565.DBX   75.0; //General Emergency Stop OK
      =     #EStopOK;

NETWORK
TITLE =read other unit's data

      SET   ;

// ... General Unit ----------/

      CALL FC   563 (
           ActReq                   := M    101.0,
           PLCNo                    := DB1565.DBW   14,
           SourceUnitNo             := 99,
           IsTUnit                  := FALSE,
           DstComDRec               := DB1565.GEN,
           RET_VAL                  := #wRetVal);


// ... CIP Unit ------------- /

      CALL FC   563 (
           ActReq                   := M    101.0,
           PLCNo                    := DB1565.DBW   14,
           SourceUnitNo             := 91,
           IsTUnit                  := FALSE,
           DstComDRec               := DB1565.CIP,
           RET_VAL                  := #wRetVal);


// ... CIP Distribution ------------- /

      L     DB1561.DBD   46;
      L     DB1945.DBD   10;
      ==D   ;
      JCN   CIP1;
      CALL FC   563 (
           ActReq                   := M    101.0,
           PLCNo                    := 3,
           SourceUnitNo             := 91,
           IsTUnit                  := FALSE,
           DstComDRec               := DB1565.CIP,
           RET_VAL                  := #wRetVal);

      CALL FC   563 (
           ActReq                   := M    101.0,
           PLCNo                    := 3,
           SourceUnitNo             := 94,
           IsTUnit                  := FALSE,
           DstComDRec               := DB1565.CIPDist,
           RET_VAL                  := #wRetVal);

      CALL SFC   20 (
           SRCBLK                   := DB1565.ToCIP,
           RET_VAL                  := #iRetVal,
           DSTBLK                   := DB502.ToCIP1);

CIP1: NOP   0;

      L     DB1561.DBD   46;
      L     DB1955.DBD   10;
      ==D   ;
      JCN   CIP2;
      CALL FC   563 (
           ActReq                   := M    101.0,
           PLCNo                    := 3,
           SourceUnitNo             := 92,
           IsTUnit                  := FALSE,
           DstComDRec               := DB1565.CIP,
           RET_VAL                  := #wRetVal);

      CALL FC   563 (
           ActReq                   := M    101.0,
           PLCNo                    := 3,
           SourceUnitNo             := 95,
           IsTUnit                  := FALSE,
           DstComDRec               := DB1565.CIPDist,
           RET_VAL                  := #wRetVal);

      CALL SFC   20 (
           SRCBLK                   := DB1565.ToCIP,
           RET_VAL                  := #iRetVal,
           DSTBLK                   := DB502.ToCIP2);
CIP2: NOP   0;

      L     DB1561.DBD   46;
      L     DB1965.DBD   10;
      ==D   ;
      JCN   CIP3;
      CALL FC   563 (
           ActReq                   := M    101.0,
           PLCNo                    := 3,
           SourceUnitNo             := 93,
           IsTUnit                  := FALSE,
           DstComDRec               := DB1565.CIP,
           RET_VAL                  := #wRetVal);

      CALL FC   563 (
           ActReq                   := M    101.0,
           PLCNo                    := 3,
           SourceUnitNo             := 96,
           IsTUnit                  := FALSE,
           DstComDRec               := DB1565.CIPDist,
           RET_VAL                  := #wRetVal);

      CALL SFC   20 (
           SRCBLK                   := DB1565.ToCIP,
           RET_VAL                  := #iRetVal,
           DSTBLK                   := DB502.ToCIP3);

CIP3: NOP   0;

//----------------------------------------
// Communication Water Tank
//----------------------------------------
// Current Tank ----------------------------
      CALL FC   950 (
           EquipmentNo              := DB1561.DBD  270,
           PLCNo                    := #iPLC,
           UnitNo                   := #iUnit);
      L     #iUnit;
      L     0;
      >I    ;
      JCN   T0xx;

      CALL FC   563 (
           ActReq                   := M    101.0,
           PLCNo                    := #iPLC,
           SourceUnitNo             := #iUnit,
           IsTUnit                  := FALSE,
           DstComDRec               := DB1565.SRC,
           RET_VAL                  := #wRetVal);
      JU    T0xy;
T0xx: NOP   0;
      T     #iTmp;
      CALL SFC   21 (
           BVAL                     := #iTmp,
           RET_VAL                  := #iRetVal,
           BLK                      := DB1565.SRC);
T0xy: NOP   0;

// Priority 1 -----------------------------
      CALL FC   950 (
           EquipmentNo              := DB1561.DBD  286,
           PLCNo                    := #iPLC,
           UnitNo                   := #iUnit);
      L     #iUnit;
      L     0;
      >I    ;
      JCN   T1xx;

      CALL FC   563 (
           ActReq                   := M    101.0,
           PLCNo                    := #iPLC,
           SourceUnitNo             := #iUnit,
           IsTUnit                  := FALSE,
           DstComDRec               := DB1565.SRC1,
           RET_VAL                  := #wRetVal);
      JU    T1xy;
T1xx: NOP   0;
      T     #iTmp;
      CALL SFC   21 (
           BVAL                     := #iTmp,
           RET_VAL                  := #iRetVal,
           BLK                      := DB1565.SRC1);
T1xy: NOP   0;

// Priority 2 ----------------------------
      CALL FC   950 (
           EquipmentNo              := DB1561.DBD  302,
           PLCNo                    := #iPLC,
           UnitNo                   := #iUnit);
      L     #iUnit;
      L     0;
      >I    ;
      JCN   T2xx;

      CALL FC   563 (
           ActReq                   := M    101.0,
           PLCNo                    := #iPLC,
           SourceUnitNo             := #iUnit,
           IsTUnit                  := FALSE,
           DstComDRec               := DB1565.SRC2,
           RET_VAL                  := #wRetVal);
      JU    T2xy;
T2xx: NOP   0;
      T     #iTmp;
      CALL SFC   21 (
           BVAL                     := #iTmp,
           RET_VAL                  := #iRetVal,
           BLK                      := DB1565.SRC2);
T2xy: NOP   0;

// Pririty 3 ----------------------------
      CALL FC   950 (
           EquipmentNo              := DB1561.DBD  318,
           PLCNo                    := #iPLC,
           UnitNo                   := #iUnit);
      L     #iUnit;
      L     0;
      >I    ;
      JCN   T3xx;

      CALL FC   563 (
           ActReq                   := M    101.0,
           PLCNo                    := #iPLC,
           SourceUnitNo             := #iUnit,
           IsTUnit                  := FALSE,
           DstComDRec               := DB1565.SRC3,
           RET_VAL                  := #wRetVal);
      JU    T3xy;
T3xx: NOP   0;
      T     #iTmp;
      CALL SFC   21 (
           BVAL                     := #iTmp,
           RET_VAL                  := #iRetVal,
           BLK                      := DB1565.SRC3);
T3xy: NOP   0;

//----------------------------------------
// Communication Fresh Water
//----------------------------------------
///   L     #U.Seq.Prop.Index0          // Destination
///   ITD
///   DTR
///   T     #rTmp

///  CALL  "Eq2PU"
//       EquipmentNo:=#rTmp
//       PLCNo      :=#iPLC
//       UnitNo     :=#iUnit

///  CALL  "UIT3"
//       ActReq      :="Clk1E"
//       PLCNo       :=#iPLC
//       SourceUnitNo:=#iUnit
//       IsTUnit     :=FALSE
//       DstComDRec  :="C04ComD".DST
//       RET_VAL     :=#wRetVal



NETWORK
TITLE =remote start

      SET   ;
// !!! insert correct condition of unit start !!!
      A     DB1561.DBX   15.0;
      A     DB1561.DBX   17.4;
      CLR   ;
      JCN   Strt;
      L     DB1565.DBD   10;
//L        L#-1;                            // Prid negative to start on its own
      T     #Prid;

      CALL FC    48 (
           UnitNo                   := #UnitNo,
           PrId                     := #Prid,
           Run                      := DB1561.DBX   17.4,
           PrIdTransfer             := TRUE,
           Start                    := TRUE,
           RetVal                   := #wRetVal);
Strt: NOP   0;
NETWORK
TITLE =external releases

      SET   ;
      =     DB2560.DBX  106.7;
NETWORK
TITLE =write own unit data

      SET   ;

//-- CIP Communication ---------------------------------------
      AN    DB1561.DBX   15.0;
//      AN "U056SeqD".Seq.PO.B30 // CIP Active (Slave)
      A     #ComCIP;
      JCN   NCIP;
//Conductivity CIP Return
      L     DB1565.DBD  150;
      T     DB1561.DBD  626;

//Temperature CIP Return
      L     DB1565.DBD  146;
      T     DB1561.DBD  594;

//CIP Prerun Pump SP

      CALL FC    45 (
           SFM                      := DB1561.DBD  686,
           Indexes                  := #SFM36);


      L     0.000000e+000;
      A     #SFM36.I01;
      =     DB1565.DBX  171.7;
      JCN   pfc;
      L     DB1561.DBD  654;
pfc:  NOP   0;
      A     #SFM36.I02;
      =     DB1565.DBX  172.0;
      JCN   ppc;
      L     DB1561.DBD  670;
ppc:  NOP   0;
      A     #SFM36.I03;
      =     DB1565.DBX  171.6;
      JCN   pxc;
      L     DB1561.DBD  574;
pxc:  NOP   0;
      T     DB1565.DBD  182;

//CIP Return
      L     DB1561.DBD  558;
      T     DB1565.DBD  186;
      L     DB1565.DBD  138;
      T     DB1561.DBD  562;

//CIP Prerun
      L     DB1561.DBD  542;
      T     DB1565.DBD  190;
      L     DB1565.DBD  142;
      T     DB1561.DBD  546;

// Write Own Data to CIP
      L     DB1565.DBD   10;
      T     DB1565.DBD  154;

      L     DB1565.DBW   14;
      T     DB1565.DBW  158;

      L     DB1565.DBW   16;
      T     DB1565.DBW  160;

      L     DB1565.DBW   18;
      T     DB1565.DBW  162;

      L     DB1565.DBW   20;
      T     DB1565.DBW  164;

      L     DB1565.DBW   22;
      T     DB1565.DBW  166;

      A     DB1565.DBX   24.0;
      =     DB1565.DBX  168.0;

      A     DB1565.DBX   24.1;
      =     DB1565.DBX  168.1;

      A     DB1565.DBX   24.2;
      =     DB1565.DBX  168.2;

      A     DB1565.DBX   24.3;
      =     DB1565.DBX  168.3;

      A     DB1565.DBX   24.4;
      =     DB1565.DBX  168.4;

      A     DB1565.DBX   24.5;
      =     DB1565.DBX  168.5;

      A     DB1565.DBX   24.6;
      =     DB1565.DBX  168.6;

      A     DB1565.DBX   24.7;
      =     DB1565.DBX  168.7;

// Copy Data to CIP
      CALL SFC   20 (
           SRCBLK                   := DB1565.ToCIP,
           RET_VAL                  := #iRetVal,
           DSTBLK                   := DB1565.ToCIP);

NCIP: NOP   0;

//Empty Signal
//A     "U056SpID".SpI.Sig //!!!! Insert correct Empty Signal !!!
      CLR   ;
      =     DB1565.DBX   26.5;

//Full Signal
//A     "U056SpID".SpI.Sig //!!!! Insert correct Full Signal !!!
      CLR   ;
      =     DB1565.DBX   26.2;

//CIP Program Selected
      A     #CIP;
      =     DB1565.DBX   27.1;

// Emergency Stop
      A     #EStopOK; //If needed add or replace with own SpI
      =     DB1565.DBX   27.0; //Emergency Stop OK

      L     DB1561.DBD  782; // Material
      T     DB1565.DBD   30;

      L     DB1561.DBD  270; // Current Water Tank Selection
      T     DB1565.DBD   34;

      L     DB1561.DBD  286; // Priority 1
      T     DB1565.DBD   38;

      L     DB1561.DBD  302; // Priority 2
      T     DB1565.DBD   42;

      L     DB1561.DBD  318; // Priority 3
      T     DB1565.DBD   46;

NETWORK
TITLE = read from other unit data



END_FUNCTION_BLOCK

FUNCTION_BLOCK FB 1569
TITLE =U056: Fresh Water Transfer
AUTHOR : Woermann
FAMILY : BOTEC_F1
NAME : Sim
VERSION : 0.1


VAR_TEMP
  CIP : BOOL ;	//CIP active
  xTmp : BOOL ;	//Temporary BOOL (free for general use)
  iTmp : INT ;	//Temporary INT (free for general use)
  rTmp : REAL ;	//Temporary REAL (free for general use)
  UnitNo : INT ;	//Unit Number
END_VAR
BEGIN
NETWORK
TITLE =General

      SET   ;
// get unit number ----------------------------------------------------------
      L     DB1560.DBW    0;
      T     #UnitNo;

// CIP ----------------------------------------------------------------------
      L     DB1561.DBD   54;
      L     0;
      <D    ;
      =     #CIP;

NETWORK
TITLE =Actuator

      A     DB1561.DBX   17.3;
      =     DB2560.DBX  105.3;
      =     DB2560.DBX  505.3;

NETWORK
TITLE =Special Input

      A     DB1561.DBX   17.3;

NETWORK
TITLE =Counter

      A     DB1561.DBX   17.3;
      A     M    101.0;


      CLR   ;
NETWORK
TITLE =Analog Input

      A     DB1561.DBX   17.3;

NETWORK
TITLE =Universal Value

      A     DB1561.DBX   17.3;
//      =     "U056UnVD".unv001.Sim;
//      =     "U056UnVD".unv002.Sim;
//      =     "U056UnVD".unv003.Sim;
//      =     "U056UnVD".unv004.Sim;

NETWORK
TITLE =PID

      A     DB1561.DBX   17.3;

NETWORK
TITLE =Message

      A     DB1561.DBX   17.3;
//      =     "U056MsgD".msg001.Sim;
//      =     "U056MsgD".msg002.Sim;
//      =     "U056MsgD".msg003.Sim;

NETWORK
TITLE =VLT

      A     DB1561.DBX   17.3;

END_FUNCTION_BLOCK

FUNCTION_BLOCK FB 1575
TITLE =U057: Water Transfer Brewhouse
FAMILY : BOTEC_F1
NAME : Comm
VERSION : 0.1


VAR_TEMP
  iRetVal : INT ;	//return value as integer
  wRetVal : WORD ;	//return value as word
  Run : BOOL ;	//Unit in "RUN" mode
  EStopOK : BOOL ;	//Emergency Stop OK
  CIP : BOOL ;	//CIP Program Selected
  ComCIP : BOOL ;	//Communication with CIP Active
  xTmp : BOOL ;	//Temporary BOOL (free for general use)
  iTmp : INT ;	//Temporary INT (free for general use)
  rTmp : REAL ;	//Temporary REAL (free for general use)
  dTmp : DINT ;	//Temporary DINT (free for general use)
  UnitNo : INT ;	//Unit Number
  EquipmentID : INT ;	//Equipment ID
  Prid : DINT ;	//Process ID
  SFM36 : STRUCT 	// CIP Pump Mode
   I00 : BOOL ;	// Off
   I01 : BOOL ;	// Flow
   I02 : BOOL ;	// Pressure
   I03 : BOOL ;	// Fix Speed
   I04 : BOOL ;
   I05 : BOOL ;
   I06 : BOOL ;
   I07 : BOOL ;
   I08 : BOOL ;
   I09 : BOOL ;
   I10 : BOOL ;
   I11 : BOOL ;
   I12 : BOOL ;
   I13 : BOOL ;
   I14 : BOOL ;
   I15 : BOOL ;
   I16 : BOOL ;
   I17 : BOOL ;
   I18 : BOOL ;
   I19 : BOOL ;
   I20 : BOOL ;
   I21 : BOOL ;
   I22 : BOOL ;
   I23 : BOOL ;
   I24 : BOOL ;
   I25 : BOOL ;
   I26 : BOOL ;
   I27 : BOOL ;
   I28 : BOOL ;
   I29 : BOOL ;
   I30 : BOOL ;
   I31 : BOOL ;
  END_STRUCT ;
  iPLC : INT ;
  iUnit : INT ;
END_VAR
BEGIN
NETWORK
TITLE =general

      SET   ;

// unit & equipment number ---------------------------------------------------
      L     DB1570.DBW    0;
      T     #UnitNo;

      L     DB1575.DBW   14;
      L     1000;
      *I    ;
      L     #UnitNo;
      +I    ;
      T     #EquipmentID;

// CIP ----------------------------------------------------------------------
      L     DB1575.DBW   18;
      L     0;
      <I    ;
      =     #CIP;

// Communicating Units-------------------------------------------------------
      L     DB1575.DBD   10;
      L     DB1575.DBD  106;
      ==D   ;
      =     #ComCIP;

// emergency OK -------------------------------------------------------------
      A     DB1575.DBX   75.0; //General Emergency Stop OK
      =     #EStopOK;

NETWORK
TITLE =read other unit's data

      SET   ;

// ... General Unit ----------/

      CALL FC   563 (
           ActReq                   := M    101.0,
           PLCNo                    := DB1575.DBW   14,
           SourceUnitNo             := 99,
           IsTUnit                  := FALSE,
           DstComDRec               := DB1575.GEN,
           RET_VAL                  := #wRetVal);


// ... CIP Unit ------------- /

